// TIA Portal V20 export
FUNCTION_BLOCK "FB_IO_Device"   // FB4, LAD
{ S7_Optimized_Access := 'TRUE' }
// stored: MemoryReserve 100, SetENOAutomatically false
   VAR_INPUT
      Test_Station : SInt;
      Life_Trigger : Bool;
      Star_Test : Bool;
      Button_Start_Approve : Bool;
      Electrical_Current_Test_Approved : Bool;
      Visual_Test_Approved : Bool;
      Electrical_Current_Read : UInt;
      Electrical_Voltage_Read : UInt;
      In_Functional_Test : "IO_Device_Functinal_Test";
      In_Test_Parameters : "IO_Device_Test_Parameters";
   END_VAR
   VAR_OUTPUT
      Reset_Functional_Test : Bool;
      Out_Test_Parameters : "IO_Device_Test_Parameters";
      Out_Functional_Test : "IO_Device_Functinal_Test";
      Out_Electrical_Voltage_Read : UInt;
   END_VAR
   VAR_TEMP   // added for the SCL form of the ladder/FBD networks
      _w1 : Bool;
   END_VAR
BEGIN

REGION Network 1: Test Parameters
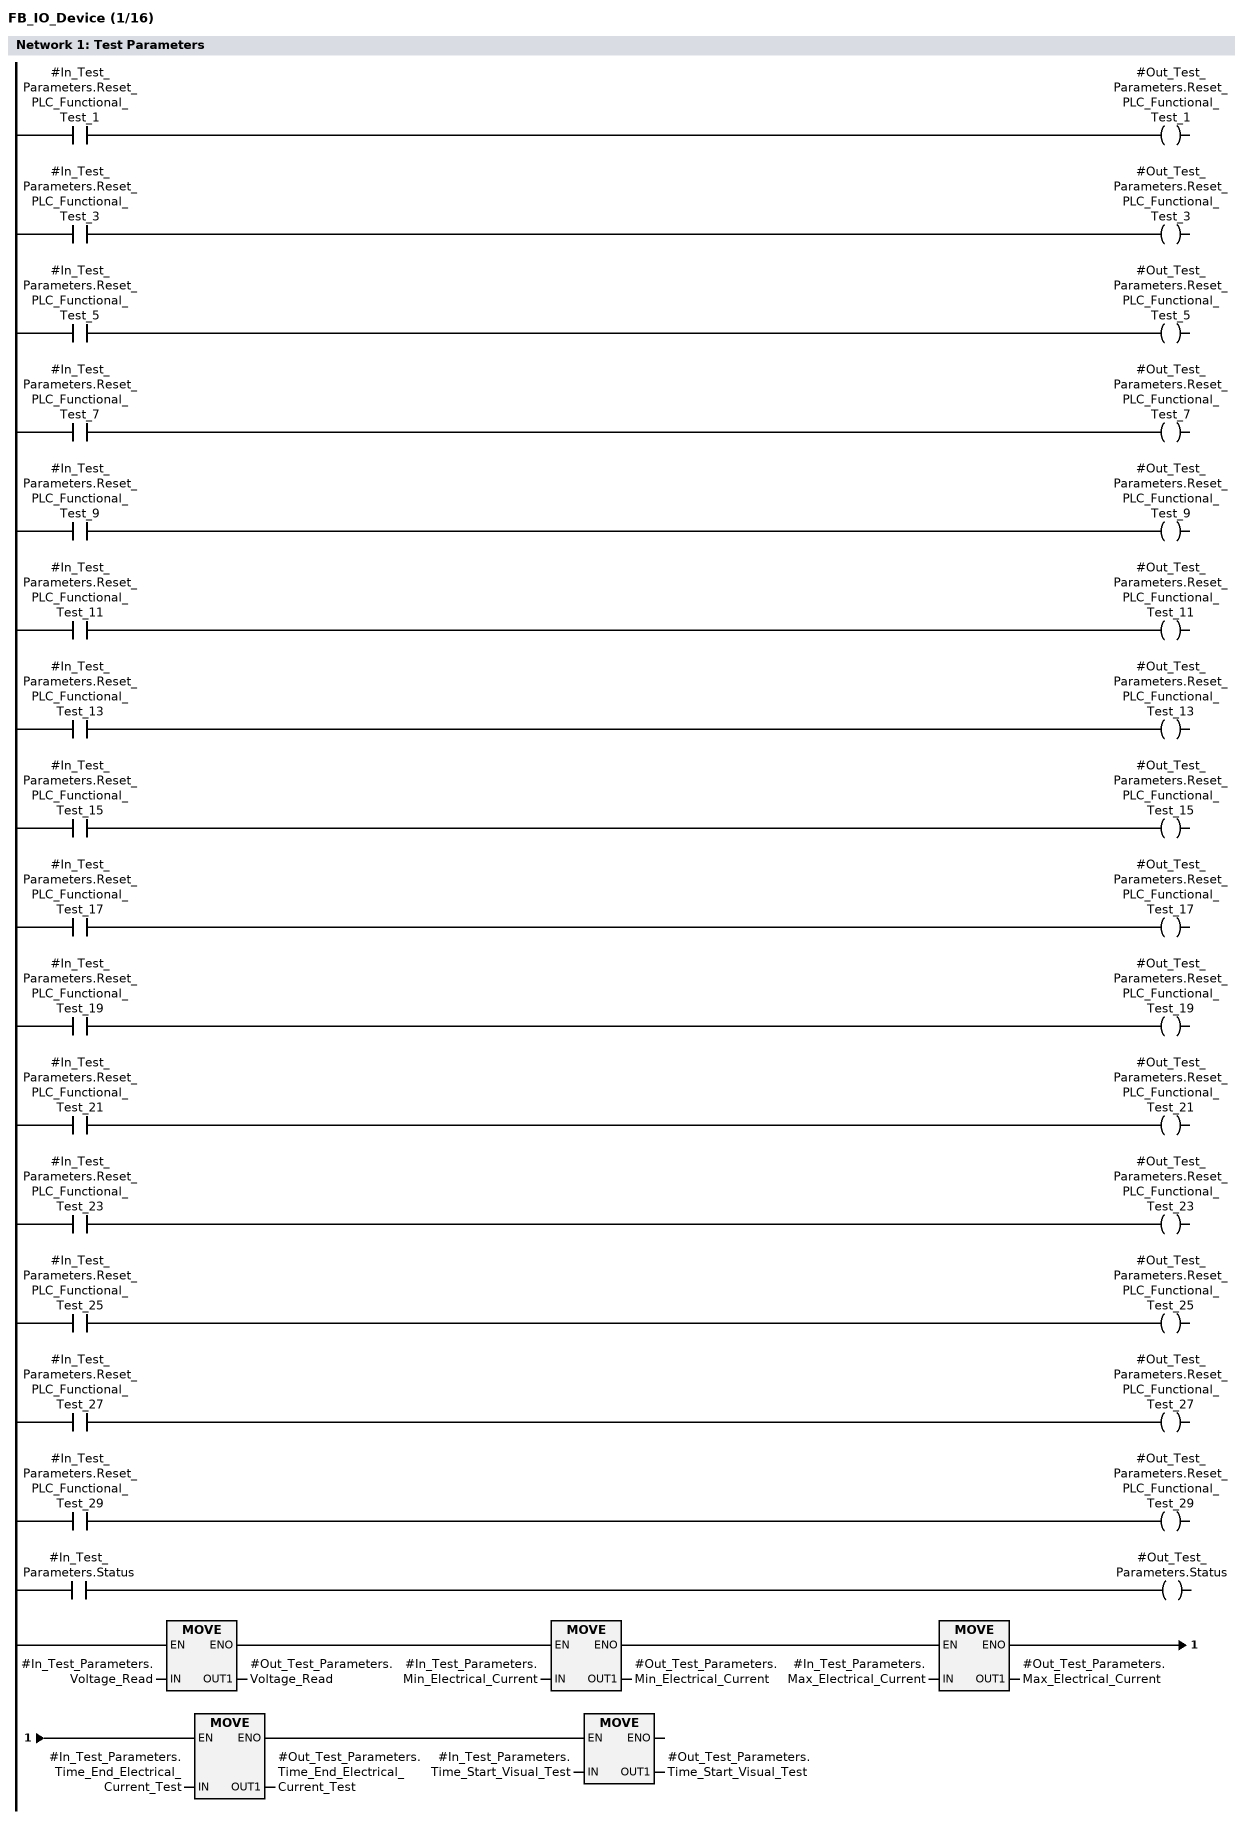
   RUNG wire#powerrail
      Contact( #In_Test_Parameters.Reset_PLC_Functional_Test_1 )
      Coil( #Out_Test_Parameters.Reset_PLC_Functional_Test_1 )
   END_RUNG
   RUNG wire#powerrail
      Contact( #In_Test_Parameters.Reset_PLC_Functional_Test_3 )
      Coil( #Out_Test_Parameters.Reset_PLC_Functional_Test_3 )
   END_RUNG
   RUNG wire#powerrail
      Contact( #In_Test_Parameters.Reset_PLC_Functional_Test_5 )
      Coil( #Out_Test_Parameters.Reset_PLC_Functional_Test_5 )
   END_RUNG
   RUNG wire#powerrail
      Contact( #In_Test_Parameters.Reset_PLC_Functional_Test_7 )
      Coil( #Out_Test_Parameters.Reset_PLC_Functional_Test_7 )
   END_RUNG
   RUNG wire#powerrail
      Contact( #In_Test_Parameters.Reset_PLC_Functional_Test_9 )
      Coil( #Out_Test_Parameters.Reset_PLC_Functional_Test_9 )
   END_RUNG
   RUNG wire#powerrail
      Contact( #In_Test_Parameters.Reset_PLC_Functional_Test_11 )
      Coil( #Out_Test_Parameters.Reset_PLC_Functional_Test_11 )
   END_RUNG
   RUNG wire#powerrail
      Contact( #In_Test_Parameters.Reset_PLC_Functional_Test_13 )
      Coil( #Out_Test_Parameters.Reset_PLC_Functional_Test_13 )
   END_RUNG
   RUNG wire#powerrail
      Contact( #In_Test_Parameters.Reset_PLC_Functional_Test_15 )
      Coil( #Out_Test_Parameters.Reset_PLC_Functional_Test_15 )
   END_RUNG
   RUNG wire#powerrail
      Contact( #In_Test_Parameters.Reset_PLC_Functional_Test_17 )
      Coil( #Out_Test_Parameters.Reset_PLC_Functional_Test_17 )
   END_RUNG
   RUNG wire#powerrail
      Contact( #In_Test_Parameters.Reset_PLC_Functional_Test_19 )
      Coil( #Out_Test_Parameters.Reset_PLC_Functional_Test_19 )
   END_RUNG
   RUNG wire#powerrail
      Contact( #In_Test_Parameters.Reset_PLC_Functional_Test_21 )
      Coil( #Out_Test_Parameters.Reset_PLC_Functional_Test_21 )
   END_RUNG
   RUNG wire#powerrail
      Contact( #In_Test_Parameters.Reset_PLC_Functional_Test_23 )
      Coil( #Out_Test_Parameters.Reset_PLC_Functional_Test_23 )
   END_RUNG
   RUNG wire#powerrail
      Contact( #In_Test_Parameters.Reset_PLC_Functional_Test_25 )
      Coil( #Out_Test_Parameters.Reset_PLC_Functional_Test_25 )
   END_RUNG
   RUNG wire#powerrail
      Contact( #In_Test_Parameters.Reset_PLC_Functional_Test_27 )
      Coil( #Out_Test_Parameters.Reset_PLC_Functional_Test_27 )
   END_RUNG
   RUNG wire#powerrail
      Contact( #In_Test_Parameters.Reset_PLC_Functional_Test_29 )
      Coil( #Out_Test_Parameters.Reset_PLC_Functional_Test_29 )
   END_RUNG
   RUNG wire#powerrail
      Contact( #In_Test_Parameters.Status )
      Coil( #Out_Test_Parameters.Status )
   END_RUNG
   RUNG wire#powerrail
      Move(in := #In_Test_Parameters.Voltage_Read, out1 => #Out_Test_Parameters.Voltage_Read)
      Move(in := #In_Test_Parameters.Min_Electrical_Current, out1 => #Out_Test_Parameters.Min_Electrical_Current)
      Move(in := #In_Test_Parameters.Max_Electrical_Current, out1 => #Out_Test_Parameters.Max_Electrical_Current)
      Move(in := #In_Test_Parameters.Time_End_Electrical_Current_Test, out1 => #Out_Test_Parameters.Time_End_Electrical_Current_Test)
      Move(in := #In_Test_Parameters.Time_Start_Visual_Test, out1 => #Out_Test_Parameters.Time_Start_Visual_Test)
   END_RUNG
   // the same network as SCL:
   #Out_Test_Parameters.Reset_PLC_Functional_Test_1 := #In_Test_Parameters.Reset_PLC_Functional_Test_1;
   #Out_Test_Parameters.Reset_PLC_Functional_Test_3 := #In_Test_Parameters.Reset_PLC_Functional_Test_3;
   #Out_Test_Parameters.Reset_PLC_Functional_Test_5 := #In_Test_Parameters.Reset_PLC_Functional_Test_5;
   #Out_Test_Parameters.Reset_PLC_Functional_Test_7 := #In_Test_Parameters.Reset_PLC_Functional_Test_7;
   #Out_Test_Parameters.Reset_PLC_Functional_Test_9 := #In_Test_Parameters.Reset_PLC_Functional_Test_9;
   #Out_Test_Parameters.Reset_PLC_Functional_Test_11 := #In_Test_Parameters.Reset_PLC_Functional_Test_11;
   #Out_Test_Parameters.Reset_PLC_Functional_Test_13 := #In_Test_Parameters.Reset_PLC_Functional_Test_13;
   #Out_Test_Parameters.Reset_PLC_Functional_Test_15 := #In_Test_Parameters.Reset_PLC_Functional_Test_15;
   #Out_Test_Parameters.Reset_PLC_Functional_Test_17 := #In_Test_Parameters.Reset_PLC_Functional_Test_17;
   #Out_Test_Parameters.Reset_PLC_Functional_Test_19 := #In_Test_Parameters.Reset_PLC_Functional_Test_19;
   #Out_Test_Parameters.Reset_PLC_Functional_Test_21 := #In_Test_Parameters.Reset_PLC_Functional_Test_21;
   #Out_Test_Parameters.Reset_PLC_Functional_Test_23 := #In_Test_Parameters.Reset_PLC_Functional_Test_23;
   #Out_Test_Parameters.Reset_PLC_Functional_Test_25 := #In_Test_Parameters.Reset_PLC_Functional_Test_25;
   #Out_Test_Parameters.Reset_PLC_Functional_Test_27 := #In_Test_Parameters.Reset_PLC_Functional_Test_27;
   #Out_Test_Parameters.Reset_PLC_Functional_Test_29 := #In_Test_Parameters.Reset_PLC_Functional_Test_29;
   #Out_Test_Parameters.Status := #In_Test_Parameters.Status;
   #Out_Test_Parameters.Voltage_Read := #In_Test_Parameters.Voltage_Read;
   #Out_Test_Parameters.Min_Electrical_Current := #In_Test_Parameters.Min_Electrical_Current;
   #Out_Test_Parameters.Max_Electrical_Current := #In_Test_Parameters.Max_Electrical_Current;
   #Out_Test_Parameters.Time_End_Electrical_Current_Test := #In_Test_Parameters.Time_End_Electrical_Current_Test;
   #Out_Test_Parameters.Time_Start_Visual_Test := #In_Test_Parameters.Time_Start_Visual_Test;
END_REGION

REGION Network 2: Functional Test Station 1
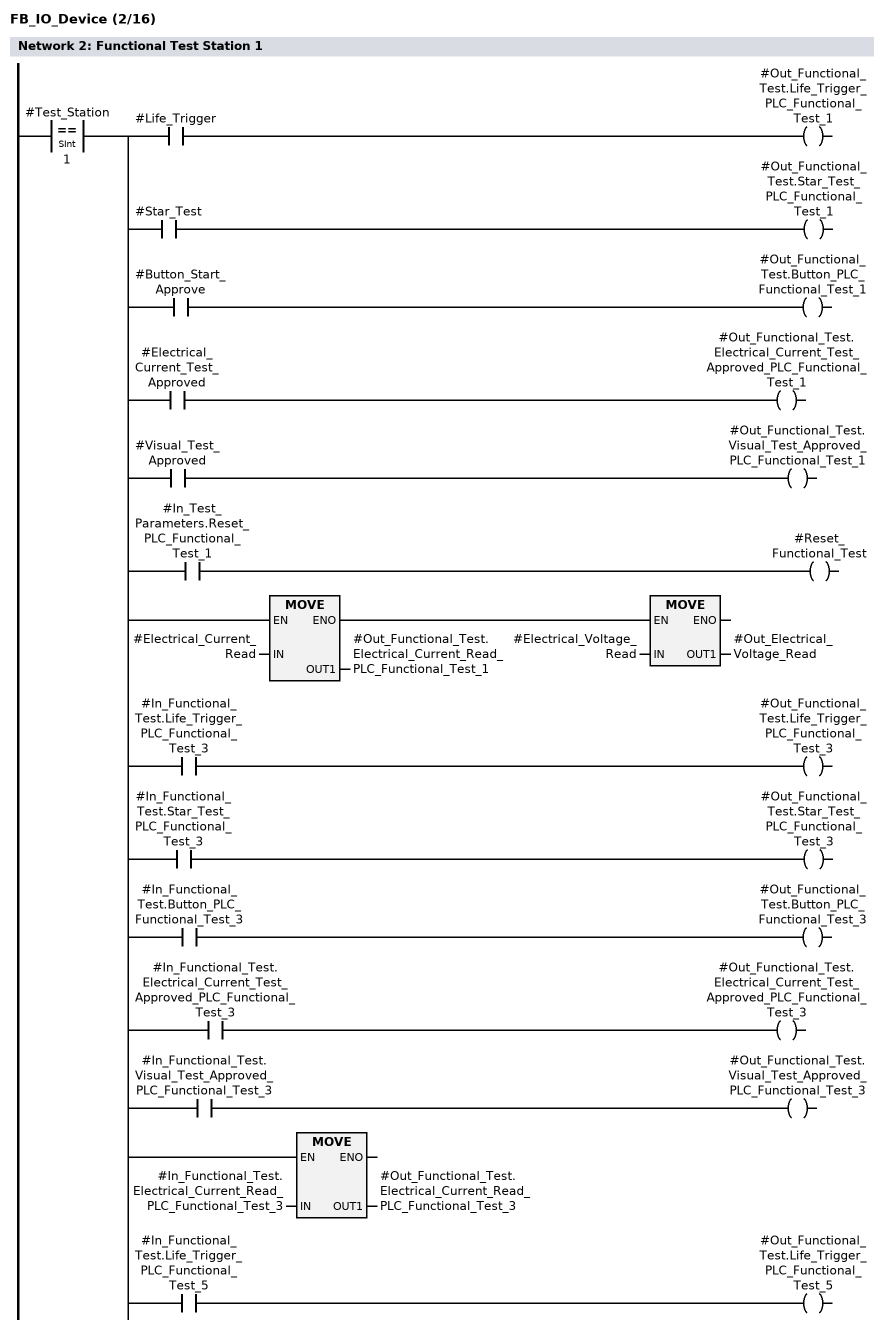
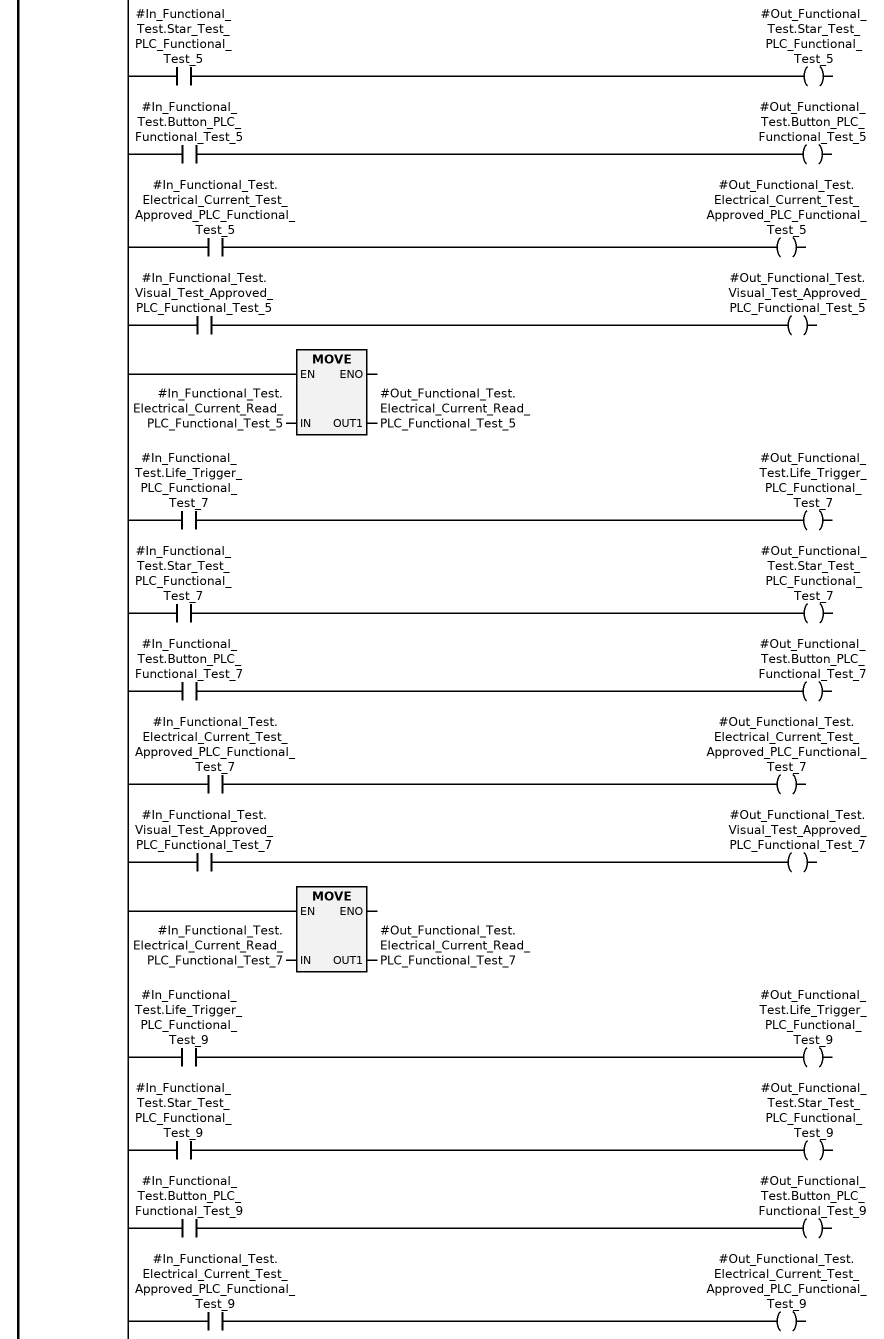
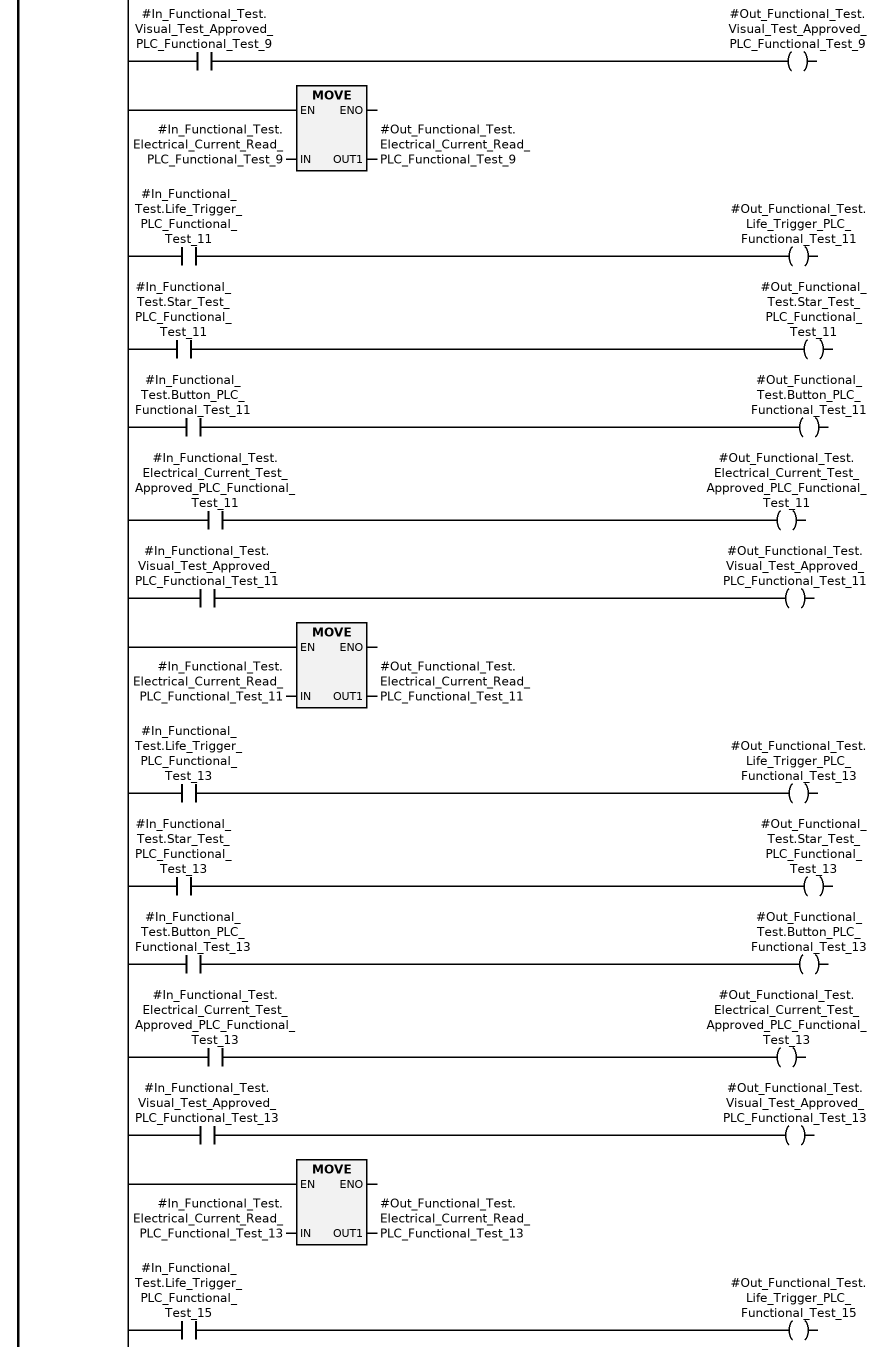
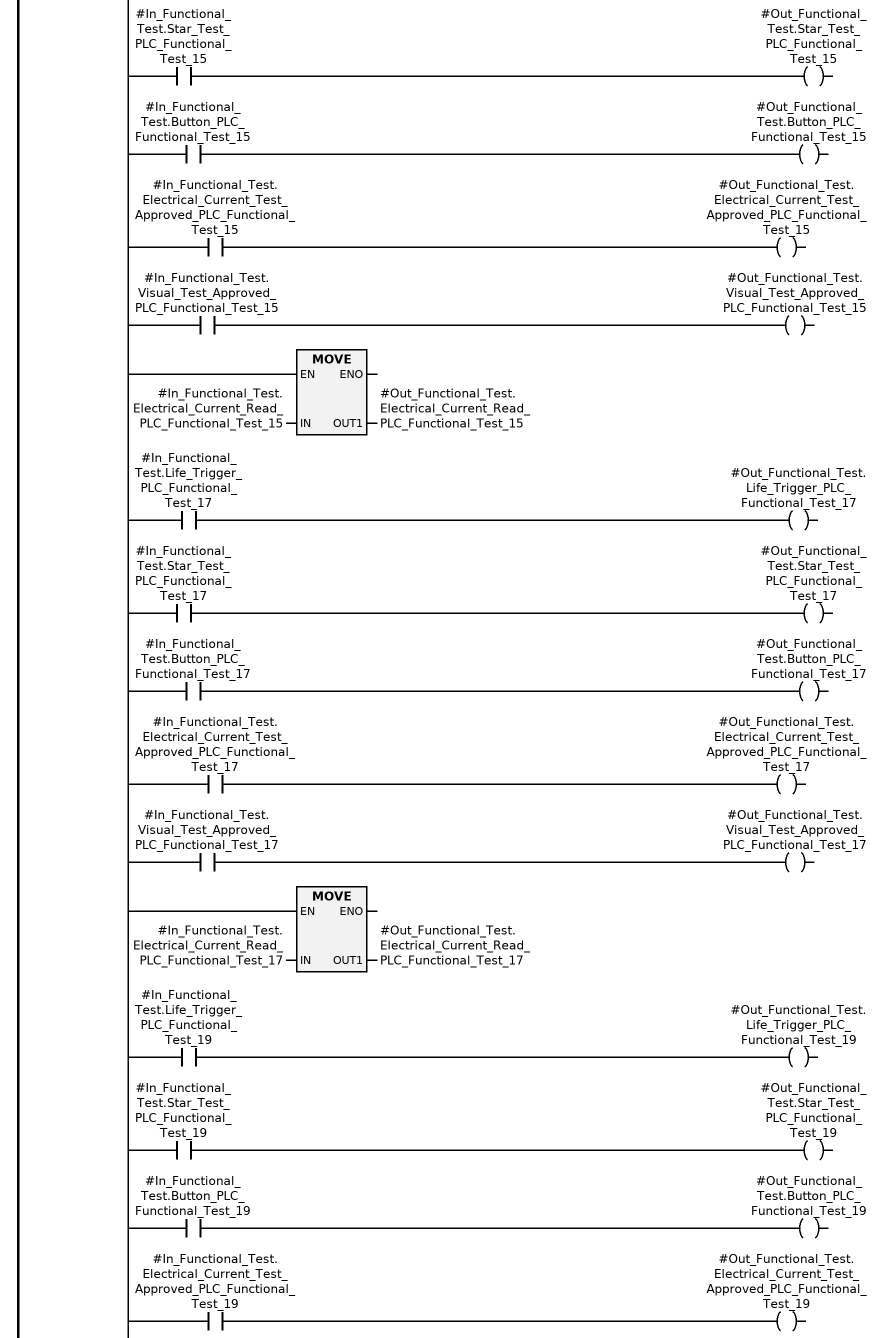
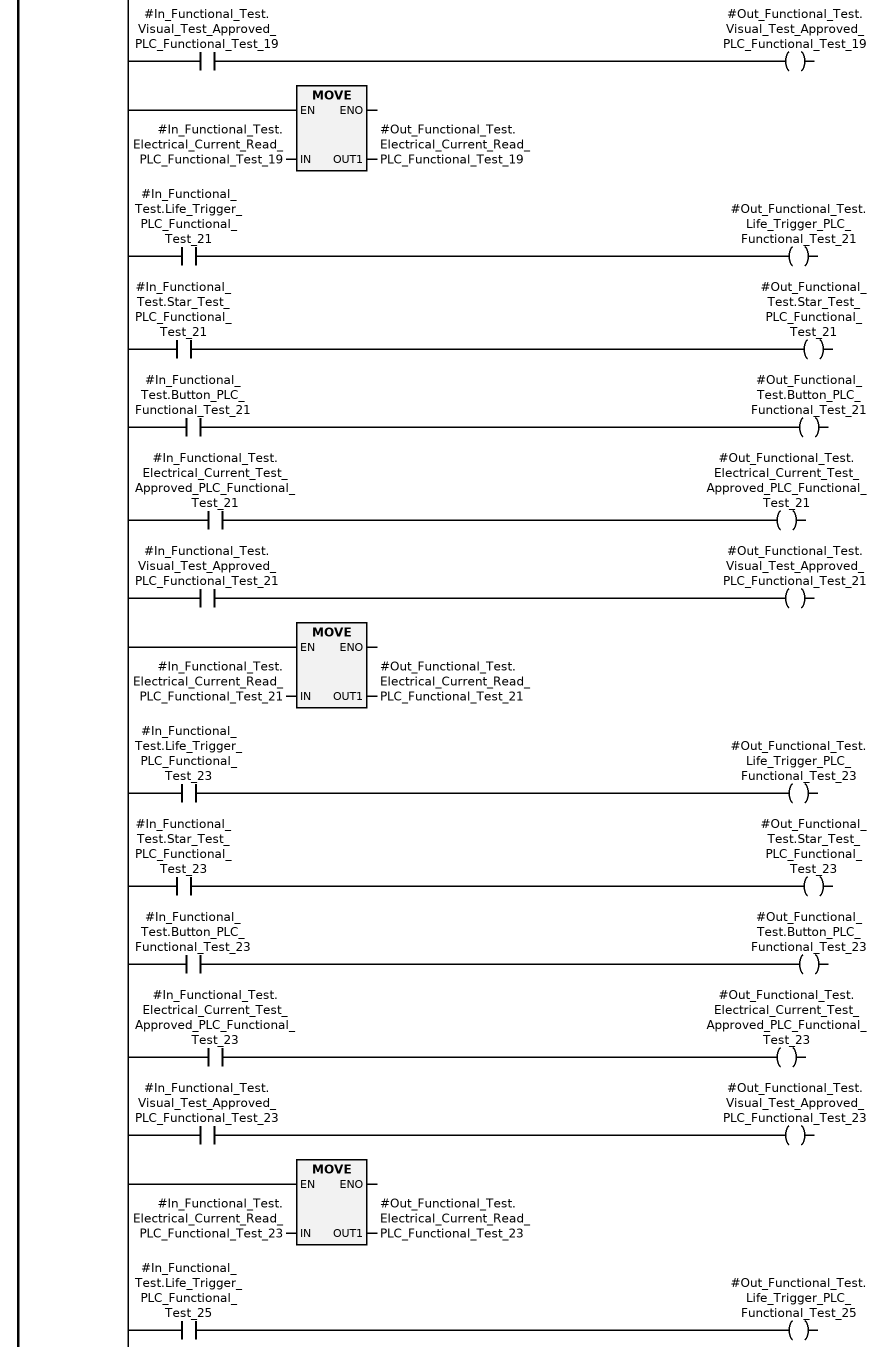
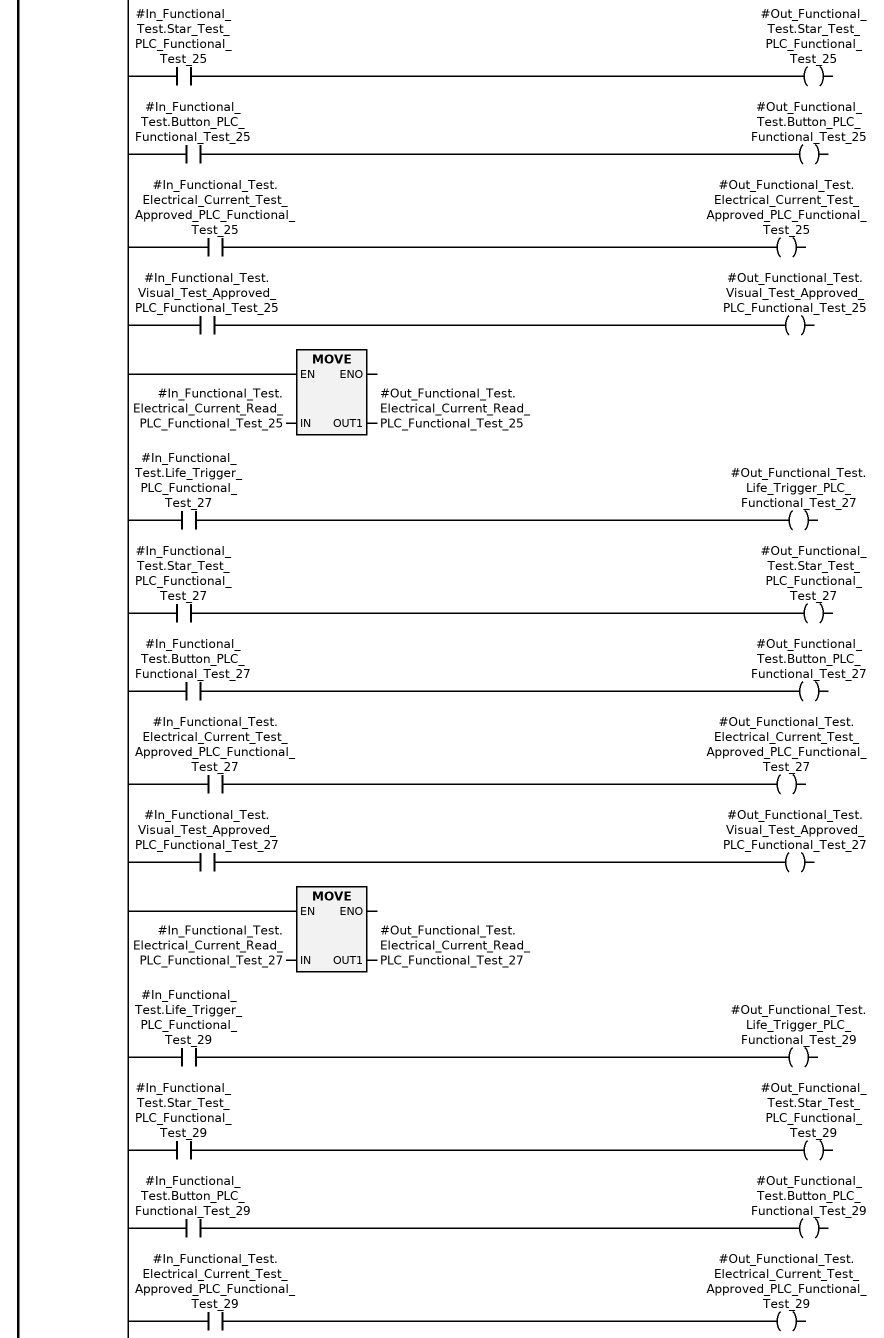
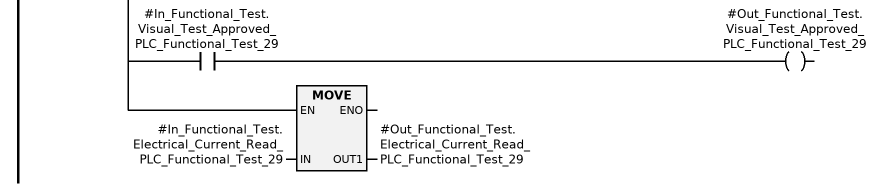
   RUNG wire#powerrail
      { S7_Templates := "SrcType := SInt" } EQ_Contact(in1 := #Test_Station, in2 := 1)
      wire#w1
      Contact( #Life_Trigger )
      Coil( #Out_Functional_Test.Life_Trigger_PLC_Functional_Test_1 )
   END_RUNG
   RUNG wire#w1
      Contact( #Star_Test )
      Coil( #Out_Functional_Test.Star_Test_PLC_Functional_Test_1 )
   END_RUNG
   RUNG wire#w1
      Contact( #Button_Start_Approve )
      Coil( #Out_Functional_Test.Button_PLC_Functional_Test_1 )
   END_RUNG
   RUNG wire#w1
      Contact( #Electrical_Current_Test_Approved )
      Coil( #Out_Functional_Test.Electrical_Current_Test_Approved_PLC_Functional_Test_1 )
   END_RUNG
   RUNG wire#w1
      Contact( #Visual_Test_Approved )
      Coil( #Out_Functional_Test.Visual_Test_Approved_PLC_Functional_Test_1 )
   END_RUNG
   RUNG wire#w1
      Contact( #In_Test_Parameters.Reset_PLC_Functional_Test_1 )
      Coil( #Reset_Functional_Test )
   END_RUNG
   RUNG wire#w1
      Move(in := #Electrical_Current_Read, out1 => #Out_Functional_Test.Electrical_Current_Read_PLC_Functional_Test_1)
      Move(in := #Electrical_Voltage_Read, out1 => #Out_Electrical_Voltage_Read)
   END_RUNG
   RUNG wire#w1
      Contact( #In_Functional_Test.Life_Trigger_PLC_Functional_Test_3 )
      Coil( #Out_Functional_Test.Life_Trigger_PLC_Functional_Test_3 )
   END_RUNG
   RUNG wire#w1
      Contact( #In_Functional_Test.Star_Test_PLC_Functional_Test_3 )
      Coil( #Out_Functional_Test.Star_Test_PLC_Functional_Test_3 )
   END_RUNG
   RUNG wire#w1
      Contact( #In_Functional_Test.Button_PLC_Functional_Test_3 )
      Coil( #Out_Functional_Test.Button_PLC_Functional_Test_3 )
   END_RUNG
   RUNG wire#w1
      Contact( #In_Functional_Test.Electrical_Current_Test_Approved_PLC_Functional_Test_3 )
      Coil( #Out_Functional_Test.Electrical_Current_Test_Approved_PLC_Functional_Test_3 )
   END_RUNG
   RUNG wire#w1
      Contact( #In_Functional_Test.Visual_Test_Approved_PLC_Functional_Test_3 )
      Coil( #Out_Functional_Test.Visual_Test_Approved_PLC_Functional_Test_3 )
   END_RUNG
   RUNG wire#w1
      Move(in := #In_Functional_Test.Electrical_Current_Read_PLC_Functional_Test_3, out1 => #Out_Functional_Test.Electrical_Current_Read_PLC_Functional_Test_3)
   END_RUNG
   RUNG wire#w1
      Contact( #In_Functional_Test.Life_Trigger_PLC_Functional_Test_5 )
      Coil( #Out_Functional_Test.Life_Trigger_PLC_Functional_Test_5 )
   END_RUNG
   RUNG wire#w1
      Contact( #In_Functional_Test.Star_Test_PLC_Functional_Test_5 )
      Coil( #Out_Functional_Test.Star_Test_PLC_Functional_Test_5 )
   END_RUNG
   RUNG wire#w1
      Contact( #In_Functional_Test.Button_PLC_Functional_Test_5 )
      Coil( #Out_Functional_Test.Button_PLC_Functional_Test_5 )
   END_RUNG
   RUNG wire#w1
      Contact( #In_Functional_Test.Electrical_Current_Test_Approved_PLC_Functional_Test_5 )
      Coil( #Out_Functional_Test.Electrical_Current_Test_Approved_PLC_Functional_Test_5 )
   END_RUNG
   RUNG wire#w1
      Contact( #In_Functional_Test.Visual_Test_Approved_PLC_Functional_Test_5 )
      Coil( #Out_Functional_Test.Visual_Test_Approved_PLC_Functional_Test_5 )
   END_RUNG
   RUNG wire#w1
      Move(in := #In_Functional_Test.Electrical_Current_Read_PLC_Functional_Test_5, out1 => #Out_Functional_Test.Electrical_Current_Read_PLC_Functional_Test_5)
   END_RUNG
   RUNG wire#w1
      Contact( #In_Functional_Test.Life_Trigger_PLC_Functional_Test_7 )
      Coil( #Out_Functional_Test.Life_Trigger_PLC_Functional_Test_7 )
   END_RUNG
   RUNG wire#w1
      Contact( #In_Functional_Test.Star_Test_PLC_Functional_Test_7 )
      Coil( #Out_Functional_Test.Star_Test_PLC_Functional_Test_7 )
   END_RUNG
   RUNG wire#w1
      Contact( #In_Functional_Test.Button_PLC_Functional_Test_7 )
      Coil( #Out_Functional_Test.Button_PLC_Functional_Test_7 )
   END_RUNG
   RUNG wire#w1
      Contact( #In_Functional_Test.Electrical_Current_Test_Approved_PLC_Functional_Test_7 )
      Coil( #Out_Functional_Test.Electrical_Current_Test_Approved_PLC_Functional_Test_7 )
   END_RUNG
   RUNG wire#w1
      Contact( #In_Functional_Test.Visual_Test_Approved_PLC_Functional_Test_7 )
      Coil( #Out_Functional_Test.Visual_Test_Approved_PLC_Functional_Test_7 )
   END_RUNG
   RUNG wire#w1
      Move(in := #In_Functional_Test.Electrical_Current_Read_PLC_Functional_Test_7, out1 => #Out_Functional_Test.Electrical_Current_Read_PLC_Functional_Test_7)
   END_RUNG
   RUNG wire#w1
      Contact( #In_Functional_Test.Life_Trigger_PLC_Functional_Test_9 )
      Coil( #Out_Functional_Test.Life_Trigger_PLC_Functional_Test_9 )
   END_RUNG
   RUNG wire#w1
      Contact( #In_Functional_Test.Star_Test_PLC_Functional_Test_9 )
      Coil( #Out_Functional_Test.Star_Test_PLC_Functional_Test_9 )
   END_RUNG
   RUNG wire#w1
      Contact( #In_Functional_Test.Button_PLC_Functional_Test_9 )
      Coil( #Out_Functional_Test.Button_PLC_Functional_Test_9 )
   END_RUNG
   RUNG wire#w1
      Contact( #In_Functional_Test.Electrical_Current_Test_Approved_PLC_Functional_Test_9 )
      Coil( #Out_Functional_Test.Electrical_Current_Test_Approved_PLC_Functional_Test_9 )
   END_RUNG
   RUNG wire#w1
      Contact( #In_Functional_Test.Visual_Test_Approved_PLC_Functional_Test_9 )
      Coil( #Out_Functional_Test.Visual_Test_Approved_PLC_Functional_Test_9 )
   END_RUNG
   RUNG wire#w1
      Move(in := #In_Functional_Test.Electrical_Current_Read_PLC_Functional_Test_9, out1 => #Out_Functional_Test.Electrical_Current_Read_PLC_Functional_Test_9)
   END_RUNG
   RUNG wire#w1
      Contact( #In_Functional_Test.Life_Trigger_PLC_Functional_Test_11 )
      Coil( #Out_Functional_Test.Life_Trigger_PLC_Functional_Test_11 )
   END_RUNG
   RUNG wire#w1
      Contact( #In_Functional_Test.Star_Test_PLC_Functional_Test_11 )
      Coil( #Out_Functional_Test.Star_Test_PLC_Functional_Test_11 )
   END_RUNG
   RUNG wire#w1
      Contact( #In_Functional_Test.Button_PLC_Functional_Test_11 )
      Coil( #Out_Functional_Test.Button_PLC_Functional_Test_11 )
   END_RUNG
   RUNG wire#w1
      Contact( #In_Functional_Test.Electrical_Current_Test_Approved_PLC_Functional_Test_11 )
      Coil( #Out_Functional_Test.Electrical_Current_Test_Approved_PLC_Functional_Test_11 )
   END_RUNG
   RUNG wire#w1
      Contact( #In_Functional_Test.Visual_Test_Approved_PLC_Functional_Test_11 )
      Coil( #Out_Functional_Test.Visual_Test_Approved_PLC_Functional_Test_11 )
   END_RUNG
   RUNG wire#w1
      Move(in := #In_Functional_Test.Electrical_Current_Read_PLC_Functional_Test_11, out1 => #Out_Functional_Test.Electrical_Current_Read_PLC_Functional_Test_11)
   END_RUNG
   RUNG wire#w1
      Contact( #In_Functional_Test.Life_Trigger_PLC_Functional_Test_13 )
      Coil( #Out_Functional_Test.Life_Trigger_PLC_Functional_Test_13 )
   END_RUNG
   RUNG wire#w1
      Contact( #In_Functional_Test.Star_Test_PLC_Functional_Test_13 )
      Coil( #Out_Functional_Test.Star_Test_PLC_Functional_Test_13 )
   END_RUNG
   RUNG wire#w1
      Contact( #In_Functional_Test.Button_PLC_Functional_Test_13 )
      Coil( #Out_Functional_Test.Button_PLC_Functional_Test_13 )
   END_RUNG
   RUNG wire#w1
      Contact( #In_Functional_Test.Electrical_Current_Test_Approved_PLC_Functional_Test_13 )
      Coil( #Out_Functional_Test.Electrical_Current_Test_Approved_PLC_Functional_Test_13 )
   END_RUNG
   RUNG wire#w1
      Contact( #In_Functional_Test.Visual_Test_Approved_PLC_Functional_Test_13 )
      Coil( #Out_Functional_Test.Visual_Test_Approved_PLC_Functional_Test_13 )
   END_RUNG
   RUNG wire#w1
      Move(in := #In_Functional_Test.Electrical_Current_Read_PLC_Functional_Test_13, out1 => #Out_Functional_Test.Electrical_Current_Read_PLC_Functional_Test_13)
   END_RUNG
   RUNG wire#w1
      Contact( #In_Functional_Test.Life_Trigger_PLC_Functional_Test_15 )
      Coil( #Out_Functional_Test.Life_Trigger_PLC_Functional_Test_15 )
   END_RUNG
   RUNG wire#w1
      Contact( #In_Functional_Test.Star_Test_PLC_Functional_Test_15 )
      Coil( #Out_Functional_Test.Star_Test_PLC_Functional_Test_15 )
   END_RUNG
   RUNG wire#w1
      Contact( #In_Functional_Test.Button_PLC_Functional_Test_15 )
      Coil( #Out_Functional_Test.Button_PLC_Functional_Test_15 )
   END_RUNG
   RUNG wire#w1
      Contact( #In_Functional_Test.Electrical_Current_Test_Approved_PLC_Functional_Test_15 )
      Coil( #Out_Functional_Test.Electrical_Current_Test_Approved_PLC_Functional_Test_15 )
   END_RUNG
   RUNG wire#w1
      Contact( #In_Functional_Test.Visual_Test_Approved_PLC_Functional_Test_15 )
      Coil( #Out_Functional_Test.Visual_Test_Approved_PLC_Functional_Test_15 )
   END_RUNG
   RUNG wire#w1
      Move(in := #In_Functional_Test.Electrical_Current_Read_PLC_Functional_Test_15, out1 => #Out_Functional_Test.Electrical_Current_Read_PLC_Functional_Test_15)
   END_RUNG
   RUNG wire#w1
      Contact( #In_Functional_Test.Life_Trigger_PLC_Functional_Test_17 )
      Coil( #Out_Functional_Test.Life_Trigger_PLC_Functional_Test_17 )
   END_RUNG
   RUNG wire#w1
      Contact( #In_Functional_Test.Star_Test_PLC_Functional_Test_17 )
      Coil( #Out_Functional_Test.Star_Test_PLC_Functional_Test_17 )
   END_RUNG
   RUNG wire#w1
      Contact( #In_Functional_Test.Button_PLC_Functional_Test_17 )
      Coil( #Out_Functional_Test.Button_PLC_Functional_Test_17 )
   END_RUNG
   RUNG wire#w1
      Contact( #In_Functional_Test.Electrical_Current_Test_Approved_PLC_Functional_Test_17 )
      Coil( #Out_Functional_Test.Electrical_Current_Test_Approved_PLC_Functional_Test_17 )
   END_RUNG
   RUNG wire#w1
      Contact( #In_Functional_Test.Visual_Test_Approved_PLC_Functional_Test_17 )
      Coil( #Out_Functional_Test.Visual_Test_Approved_PLC_Functional_Test_17 )
   END_RUNG
   RUNG wire#w1
      Move(in := #In_Functional_Test.Electrical_Current_Read_PLC_Functional_Test_17, out1 => #Out_Functional_Test.Electrical_Current_Read_PLC_Functional_Test_17)
   END_RUNG
   RUNG wire#w1
      Contact( #In_Functional_Test.Life_Trigger_PLC_Functional_Test_19 )
      Coil( #Out_Functional_Test.Life_Trigger_PLC_Functional_Test_19 )
   END_RUNG
   RUNG wire#w1
      Contact( #In_Functional_Test.Star_Test_PLC_Functional_Test_19 )
      Coil( #Out_Functional_Test.Star_Test_PLC_Functional_Test_19 )
   END_RUNG
   RUNG wire#w1
      Contact( #In_Functional_Test.Button_PLC_Functional_Test_19 )
      Coil( #Out_Functional_Test.Button_PLC_Functional_Test_19 )
   END_RUNG
   RUNG wire#w1
      Contact( #In_Functional_Test.Electrical_Current_Test_Approved_PLC_Functional_Test_19 )
      Coil( #Out_Functional_Test.Electrical_Current_Test_Approved_PLC_Functional_Test_19 )
   END_RUNG
   RUNG wire#w1
      Contact( #In_Functional_Test.Visual_Test_Approved_PLC_Functional_Test_19 )
      Coil( #Out_Functional_Test.Visual_Test_Approved_PLC_Functional_Test_19 )
   END_RUNG
   RUNG wire#w1
      Move(in := #In_Functional_Test.Electrical_Current_Read_PLC_Functional_Test_19, out1 => #Out_Functional_Test.Electrical_Current_Read_PLC_Functional_Test_19)
   END_RUNG
   RUNG wire#w1
      Contact( #In_Functional_Test.Life_Trigger_PLC_Functional_Test_21 )
      Coil( #Out_Functional_Test.Life_Trigger_PLC_Functional_Test_21 )
   END_RUNG
   RUNG wire#w1
      Contact( #In_Functional_Test.Star_Test_PLC_Functional_Test_21 )
      Coil( #Out_Functional_Test.Star_Test_PLC_Functional_Test_21 )
   END_RUNG
   RUNG wire#w1
      Contact( #In_Functional_Test.Button_PLC_Functional_Test_21 )
      Coil( #Out_Functional_Test.Button_PLC_Functional_Test_21 )
   END_RUNG
   RUNG wire#w1
      Contact( #In_Functional_Test.Electrical_Current_Test_Approved_PLC_Functional_Test_21 )
      Coil( #Out_Functional_Test.Electrical_Current_Test_Approved_PLC_Functional_Test_21 )
   END_RUNG
   RUNG wire#w1
      Contact( #In_Functional_Test.Visual_Test_Approved_PLC_Functional_Test_21 )
      Coil( #Out_Functional_Test.Visual_Test_Approved_PLC_Functional_Test_21 )
   END_RUNG
   RUNG wire#w1
      Move(in := #In_Functional_Test.Electrical_Current_Read_PLC_Functional_Test_21, out1 => #Out_Functional_Test.Electrical_Current_Read_PLC_Functional_Test_21)
   END_RUNG
   RUNG wire#w1
      Contact( #In_Functional_Test.Life_Trigger_PLC_Functional_Test_23 )
      Coil( #Out_Functional_Test.Life_Trigger_PLC_Functional_Test_23 )
   END_RUNG
   RUNG wire#w1
      Contact( #In_Functional_Test.Star_Test_PLC_Functional_Test_23 )
      Coil( #Out_Functional_Test.Star_Test_PLC_Functional_Test_23 )
   END_RUNG
   RUNG wire#w1
      Contact( #In_Functional_Test.Button_PLC_Functional_Test_23 )
      Coil( #Out_Functional_Test.Button_PLC_Functional_Test_23 )
   END_RUNG
   RUNG wire#w1
      Contact( #In_Functional_Test.Electrical_Current_Test_Approved_PLC_Functional_Test_23 )
      Coil( #Out_Functional_Test.Electrical_Current_Test_Approved_PLC_Functional_Test_23 )
   END_RUNG
   RUNG wire#w1
      Contact( #In_Functional_Test.Visual_Test_Approved_PLC_Functional_Test_23 )
      Coil( #Out_Functional_Test.Visual_Test_Approved_PLC_Functional_Test_23 )
   END_RUNG
   RUNG wire#w1
      Move(in := #In_Functional_Test.Electrical_Current_Read_PLC_Functional_Test_23, out1 => #Out_Functional_Test.Electrical_Current_Read_PLC_Functional_Test_23)
   END_RUNG
   RUNG wire#w1
      Contact( #In_Functional_Test.Life_Trigger_PLC_Functional_Test_25 )
      Coil( #Out_Functional_Test.Life_Trigger_PLC_Functional_Test_25 )
   END_RUNG
   RUNG wire#w1
      Contact( #In_Functional_Test.Star_Test_PLC_Functional_Test_25 )
      Coil( #Out_Functional_Test.Star_Test_PLC_Functional_Test_25 )
   END_RUNG
   RUNG wire#w1
      Contact( #In_Functional_Test.Button_PLC_Functional_Test_25 )
      Coil( #Out_Functional_Test.Button_PLC_Functional_Test_25 )
   END_RUNG
   RUNG wire#w1
      Contact( #In_Functional_Test.Electrical_Current_Test_Approved_PLC_Functional_Test_25 )
      Coil( #Out_Functional_Test.Electrical_Current_Test_Approved_PLC_Functional_Test_25 )
   END_RUNG
   RUNG wire#w1
      Contact( #In_Functional_Test.Visual_Test_Approved_PLC_Functional_Test_25 )
      Coil( #Out_Functional_Test.Visual_Test_Approved_PLC_Functional_Test_25 )
   END_RUNG
   RUNG wire#w1
      Move(in := #In_Functional_Test.Electrical_Current_Read_PLC_Functional_Test_25, out1 => #Out_Functional_Test.Electrical_Current_Read_PLC_Functional_Test_25)
   END_RUNG
   RUNG wire#w1
      Contact( #In_Functional_Test.Life_Trigger_PLC_Functional_Test_27 )
      Coil( #Out_Functional_Test.Life_Trigger_PLC_Functional_Test_27 )
   END_RUNG
   RUNG wire#w1
      Contact( #In_Functional_Test.Star_Test_PLC_Functional_Test_27 )
      Coil( #Out_Functional_Test.Star_Test_PLC_Functional_Test_27 )
   END_RUNG
   RUNG wire#w1
      Contact( #In_Functional_Test.Button_PLC_Functional_Test_27 )
      Coil( #Out_Functional_Test.Button_PLC_Functional_Test_27 )
   END_RUNG
   RUNG wire#w1
      Contact( #In_Functional_Test.Electrical_Current_Test_Approved_PLC_Functional_Test_27 )
      Coil( #Out_Functional_Test.Electrical_Current_Test_Approved_PLC_Functional_Test_27 )
   END_RUNG
   RUNG wire#w1
      Contact( #In_Functional_Test.Visual_Test_Approved_PLC_Functional_Test_27 )
      Coil( #Out_Functional_Test.Visual_Test_Approved_PLC_Functional_Test_27 )
   END_RUNG
   RUNG wire#w1
      Move(in := #In_Functional_Test.Electrical_Current_Read_PLC_Functional_Test_27, out1 => #Out_Functional_Test.Electrical_Current_Read_PLC_Functional_Test_27)
   END_RUNG
   RUNG wire#w1
      Contact( #In_Functional_Test.Life_Trigger_PLC_Functional_Test_29 )
      Coil( #Out_Functional_Test.Life_Trigger_PLC_Functional_Test_29 )
   END_RUNG
   RUNG wire#w1
      Contact( #In_Functional_Test.Star_Test_PLC_Functional_Test_29 )
      Coil( #Out_Functional_Test.Star_Test_PLC_Functional_Test_29 )
   END_RUNG
   RUNG wire#w1
      Contact( #In_Functional_Test.Button_PLC_Functional_Test_29 )
      Coil( #Out_Functional_Test.Button_PLC_Functional_Test_29 )
   END_RUNG
   RUNG wire#w1
      Contact( #In_Functional_Test.Electrical_Current_Test_Approved_PLC_Functional_Test_29 )
      Coil( #Out_Functional_Test.Electrical_Current_Test_Approved_PLC_Functional_Test_29 )
   END_RUNG
   RUNG wire#w1
      Contact( #In_Functional_Test.Visual_Test_Approved_PLC_Functional_Test_29 )
      Coil( #Out_Functional_Test.Visual_Test_Approved_PLC_Functional_Test_29 )
   END_RUNG
   RUNG wire#w1
      Move(in := #In_Functional_Test.Electrical_Current_Read_PLC_Functional_Test_29, out1 => #Out_Functional_Test.Electrical_Current_Read_PLC_Functional_Test_29)
   END_RUNG
   // the same network as SCL:
   #_w1 := #Test_Station = 1;
   #Out_Functional_Test.Life_Trigger_PLC_Functional_Test_1 := #_w1 AND #Life_Trigger;
   #Out_Functional_Test.Star_Test_PLC_Functional_Test_1 := #_w1 AND #Star_Test;
   #Out_Functional_Test.Button_PLC_Functional_Test_1 := #_w1 AND #Button_Start_Approve;
   #Out_Functional_Test.Electrical_Current_Test_Approved_PLC_Functional_Test_1 := #_w1 AND #Electrical_Current_Test_Approved;
   #Out_Functional_Test.Visual_Test_Approved_PLC_Functional_Test_1 := #_w1 AND #Visual_Test_Approved;
   #Reset_Functional_Test := #_w1 AND #In_Test_Parameters.Reset_PLC_Functional_Test_1;
   IF #_w1 THEN
       #Out_Functional_Test.Electrical_Current_Read_PLC_Functional_Test_1 := #Electrical_Current_Read;
       #Out_Electrical_Voltage_Read := #Electrical_Voltage_Read;
   END_IF;
   #Out_Functional_Test.Life_Trigger_PLC_Functional_Test_3 := #_w1 AND #In_Functional_Test.Life_Trigger_PLC_Functional_Test_3;
   #Out_Functional_Test.Star_Test_PLC_Functional_Test_3 := #_w1 AND #In_Functional_Test.Star_Test_PLC_Functional_Test_3;
   #Out_Functional_Test.Button_PLC_Functional_Test_3 := #_w1 AND #In_Functional_Test.Button_PLC_Functional_Test_3;
   #Out_Functional_Test.Electrical_Current_Test_Approved_PLC_Functional_Test_3 := #_w1 AND #In_Functional_Test.Electrical_Current_Test_Approved_PLC_Functional_Test_3;
   #Out_Functional_Test.Visual_Test_Approved_PLC_Functional_Test_3 := #_w1 AND #In_Functional_Test.Visual_Test_Approved_PLC_Functional_Test_3;
   IF #_w1 THEN
       #Out_Functional_Test.Electrical_Current_Read_PLC_Functional_Test_3 := #In_Functional_Test.Electrical_Current_Read_PLC_Functional_Test_3;
   END_IF;
   #Out_Functional_Test.Life_Trigger_PLC_Functional_Test_5 := #_w1 AND #In_Functional_Test.Life_Trigger_PLC_Functional_Test_5;
   #Out_Functional_Test.Star_Test_PLC_Functional_Test_5 := #_w1 AND #In_Functional_Test.Star_Test_PLC_Functional_Test_5;
   #Out_Functional_Test.Button_PLC_Functional_Test_5 := #_w1 AND #In_Functional_Test.Button_PLC_Functional_Test_5;
   #Out_Functional_Test.Electrical_Current_Test_Approved_PLC_Functional_Test_5 := #_w1 AND #In_Functional_Test.Electrical_Current_Test_Approved_PLC_Functional_Test_5;
   #Out_Functional_Test.Visual_Test_Approved_PLC_Functional_Test_5 := #_w1 AND #In_Functional_Test.Visual_Test_Approved_PLC_Functional_Test_5;
   IF #_w1 THEN
       #Out_Functional_Test.Electrical_Current_Read_PLC_Functional_Test_5 := #In_Functional_Test.Electrical_Current_Read_PLC_Functional_Test_5;
   END_IF;
   #Out_Functional_Test.Life_Trigger_PLC_Functional_Test_7 := #_w1 AND #In_Functional_Test.Life_Trigger_PLC_Functional_Test_7;
   #Out_Functional_Test.Star_Test_PLC_Functional_Test_7 := #_w1 AND #In_Functional_Test.Star_Test_PLC_Functional_Test_7;
   #Out_Functional_Test.Button_PLC_Functional_Test_7 := #_w1 AND #In_Functional_Test.Button_PLC_Functional_Test_7;
   #Out_Functional_Test.Electrical_Current_Test_Approved_PLC_Functional_Test_7 := #_w1 AND #In_Functional_Test.Electrical_Current_Test_Approved_PLC_Functional_Test_7;
   #Out_Functional_Test.Visual_Test_Approved_PLC_Functional_Test_7 := #_w1 AND #In_Functional_Test.Visual_Test_Approved_PLC_Functional_Test_7;
   IF #_w1 THEN
       #Out_Functional_Test.Electrical_Current_Read_PLC_Functional_Test_7 := #In_Functional_Test.Electrical_Current_Read_PLC_Functional_Test_7;
   END_IF;
   #Out_Functional_Test.Life_Trigger_PLC_Functional_Test_9 := #_w1 AND #In_Functional_Test.Life_Trigger_PLC_Functional_Test_9;
   #Out_Functional_Test.Star_Test_PLC_Functional_Test_9 := #_w1 AND #In_Functional_Test.Star_Test_PLC_Functional_Test_9;
   #Out_Functional_Test.Button_PLC_Functional_Test_9 := #_w1 AND #In_Functional_Test.Button_PLC_Functional_Test_9;
   #Out_Functional_Test.Electrical_Current_Test_Approved_PLC_Functional_Test_9 := #_w1 AND #In_Functional_Test.Electrical_Current_Test_Approved_PLC_Functional_Test_9;
   #Out_Functional_Test.Visual_Test_Approved_PLC_Functional_Test_9 := #_w1 AND #In_Functional_Test.Visual_Test_Approved_PLC_Functional_Test_9;
   IF #_w1 THEN
       #Out_Functional_Test.Electrical_Current_Read_PLC_Functional_Test_9 := #In_Functional_Test.Electrical_Current_Read_PLC_Functional_Test_9;
   END_IF;
   #Out_Functional_Test.Life_Trigger_PLC_Functional_Test_11 := #_w1 AND #In_Functional_Test.Life_Trigger_PLC_Functional_Test_11;
   #Out_Functional_Test.Star_Test_PLC_Functional_Test_11 := #_w1 AND #In_Functional_Test.Star_Test_PLC_Functional_Test_11;
   #Out_Functional_Test.Button_PLC_Functional_Test_11 := #_w1 AND #In_Functional_Test.Button_PLC_Functional_Test_11;
   #Out_Functional_Test.Electrical_Current_Test_Approved_PLC_Functional_Test_11 := #_w1 AND #In_Functional_Test.Electrical_Current_Test_Approved_PLC_Functional_Test_11;
   #Out_Functional_Test.Visual_Test_Approved_PLC_Functional_Test_11 := #_w1 AND #In_Functional_Test.Visual_Test_Approved_PLC_Functional_Test_11;
   IF #_w1 THEN
       #Out_Functional_Test.Electrical_Current_Read_PLC_Functional_Test_11 := #In_Functional_Test.Electrical_Current_Read_PLC_Functional_Test_11;
   END_IF;
   #Out_Functional_Test.Life_Trigger_PLC_Functional_Test_13 := #_w1 AND #In_Functional_Test.Life_Trigger_PLC_Functional_Test_13;
   #Out_Functional_Test.Star_Test_PLC_Functional_Test_13 := #_w1 AND #In_Functional_Test.Star_Test_PLC_Functional_Test_13;
   #Out_Functional_Test.Button_PLC_Functional_Test_13 := #_w1 AND #In_Functional_Test.Button_PLC_Functional_Test_13;
   #Out_Functional_Test.Electrical_Current_Test_Approved_PLC_Functional_Test_13 := #_w1 AND #In_Functional_Test.Electrical_Current_Test_Approved_PLC_Functional_Test_13;
   #Out_Functional_Test.Visual_Test_Approved_PLC_Functional_Test_13 := #_w1 AND #In_Functional_Test.Visual_Test_Approved_PLC_Functional_Test_13;
   IF #_w1 THEN
       #Out_Functional_Test.Electrical_Current_Read_PLC_Functional_Test_13 := #In_Functional_Test.Electrical_Current_Read_PLC_Functional_Test_13;
   END_IF;
   #Out_Functional_Test.Life_Trigger_PLC_Functional_Test_15 := #_w1 AND #In_Functional_Test.Life_Trigger_PLC_Functional_Test_15;
   #Out_Functional_Test.Star_Test_PLC_Functional_Test_15 := #_w1 AND #In_Functional_Test.Star_Test_PLC_Functional_Test_15;
   #Out_Functional_Test.Button_PLC_Functional_Test_15 := #_w1 AND #In_Functional_Test.Button_PLC_Functional_Test_15;
   #Out_Functional_Test.Electrical_Current_Test_Approved_PLC_Functional_Test_15 := #_w1 AND #In_Functional_Test.Electrical_Current_Test_Approved_PLC_Functional_Test_15;
   #Out_Functional_Test.Visual_Test_Approved_PLC_Functional_Test_15 := #_w1 AND #In_Functional_Test.Visual_Test_Approved_PLC_Functional_Test_15;
   IF #_w1 THEN
       #Out_Functional_Test.Electrical_Current_Read_PLC_Functional_Test_15 := #In_Functional_Test.Electrical_Current_Read_PLC_Functional_Test_15;
   END_IF;
   #Out_Functional_Test.Life_Trigger_PLC_Functional_Test_17 := #_w1 AND #In_Functional_Test.Life_Trigger_PLC_Functional_Test_17;
   #Out_Functional_Test.Star_Test_PLC_Functional_Test_17 := #_w1 AND #In_Functional_Test.Star_Test_PLC_Functional_Test_17;
   #Out_Functional_Test.Button_PLC_Functional_Test_17 := #_w1 AND #In_Functional_Test.Button_PLC_Functional_Test_17;
   #Out_Functional_Test.Electrical_Current_Test_Approved_PLC_Functional_Test_17 := #_w1 AND #In_Functional_Test.Electrical_Current_Test_Approved_PLC_Functional_Test_17;
   #Out_Functional_Test.Visual_Test_Approved_PLC_Functional_Test_17 := #_w1 AND #In_Functional_Test.Visual_Test_Approved_PLC_Functional_Test_17;
   IF #_w1 THEN
       #Out_Functional_Test.Electrical_Current_Read_PLC_Functional_Test_17 := #In_Functional_Test.Electrical_Current_Read_PLC_Functional_Test_17;
   END_IF;
   #Out_Functional_Test.Life_Trigger_PLC_Functional_Test_19 := #_w1 AND #In_Functional_Test.Life_Trigger_PLC_Functional_Test_19;
   #Out_Functional_Test.Star_Test_PLC_Functional_Test_19 := #_w1 AND #In_Functional_Test.Star_Test_PLC_Functional_Test_19;
   #Out_Functional_Test.Button_PLC_Functional_Test_19 := #_w1 AND #In_Functional_Test.Button_PLC_Functional_Test_19;
   #Out_Functional_Test.Electrical_Current_Test_Approved_PLC_Functional_Test_19 := #_w1 AND #In_Functional_Test.Electrical_Current_Test_Approved_PLC_Functional_Test_19;
   #Out_Functional_Test.Visual_Test_Approved_PLC_Functional_Test_19 := #_w1 AND #In_Functional_Test.Visual_Test_Approved_PLC_Functional_Test_19;
   IF #_w1 THEN
       #Out_Functional_Test.Electrical_Current_Read_PLC_Functional_Test_19 := #In_Functional_Test.Electrical_Current_Read_PLC_Functional_Test_19;
   END_IF;
   #Out_Functional_Test.Life_Trigger_PLC_Functional_Test_21 := #_w1 AND #In_Functional_Test.Life_Trigger_PLC_Functional_Test_21;
   #Out_Functional_Test.Star_Test_PLC_Functional_Test_21 := #_w1 AND #In_Functional_Test.Star_Test_PLC_Functional_Test_21;
   #Out_Functional_Test.Button_PLC_Functional_Test_21 := #_w1 AND #In_Functional_Test.Button_PLC_Functional_Test_21;
   #Out_Functional_Test.Electrical_Current_Test_Approved_PLC_Functional_Test_21 := #_w1 AND #In_Functional_Test.Electrical_Current_Test_Approved_PLC_Functional_Test_21;
   #Out_Functional_Test.Visual_Test_Approved_PLC_Functional_Test_21 := #_w1 AND #In_Functional_Test.Visual_Test_Approved_PLC_Functional_Test_21;
   IF #_w1 THEN
       #Out_Functional_Test.Electrical_Current_Read_PLC_Functional_Test_21 := #In_Functional_Test.Electrical_Current_Read_PLC_Functional_Test_21;
   END_IF;
   #Out_Functional_Test.Life_Trigger_PLC_Functional_Test_23 := #_w1 AND #In_Functional_Test.Life_Trigger_PLC_Functional_Test_23;
   #Out_Functional_Test.Star_Test_PLC_Functional_Test_23 := #_w1 AND #In_Functional_Test.Star_Test_PLC_Functional_Test_23;
   #Out_Functional_Test.Button_PLC_Functional_Test_23 := #_w1 AND #In_Functional_Test.Button_PLC_Functional_Test_23;
   #Out_Functional_Test.Electrical_Current_Test_Approved_PLC_Functional_Test_23 := #_w1 AND #In_Functional_Test.Electrical_Current_Test_Approved_PLC_Functional_Test_23;
   #Out_Functional_Test.Visual_Test_Approved_PLC_Functional_Test_23 := #_w1 AND #In_Functional_Test.Visual_Test_Approved_PLC_Functional_Test_23;
   IF #_w1 THEN
       #Out_Functional_Test.Electrical_Current_Read_PLC_Functional_Test_23 := #In_Functional_Test.Electrical_Current_Read_PLC_Functional_Test_23;
   END_IF;
   #Out_Functional_Test.Life_Trigger_PLC_Functional_Test_25 := #_w1 AND #In_Functional_Test.Life_Trigger_PLC_Functional_Test_25;
   #Out_Functional_Test.Star_Test_PLC_Functional_Test_25 := #_w1 AND #In_Functional_Test.Star_Test_PLC_Functional_Test_25;
   #Out_Functional_Test.Button_PLC_Functional_Test_25 := #_w1 AND #In_Functional_Test.Button_PLC_Functional_Test_25;
   #Out_Functional_Test.Electrical_Current_Test_Approved_PLC_Functional_Test_25 := #_w1 AND #In_Functional_Test.Electrical_Current_Test_Approved_PLC_Functional_Test_25;
   #Out_Functional_Test.Visual_Test_Approved_PLC_Functional_Test_25 := #_w1 AND #In_Functional_Test.Visual_Test_Approved_PLC_Functional_Test_25;
   IF #_w1 THEN
       #Out_Functional_Test.Electrical_Current_Read_PLC_Functional_Test_25 := #In_Functional_Test.Electrical_Current_Read_PLC_Functional_Test_25;
   END_IF;
   #Out_Functional_Test.Life_Trigger_PLC_Functional_Test_27 := #_w1 AND #In_Functional_Test.Life_Trigger_PLC_Functional_Test_27;
   #Out_Functional_Test.Star_Test_PLC_Functional_Test_27 := #_w1 AND #In_Functional_Test.Star_Test_PLC_Functional_Test_27;
   #Out_Functional_Test.Button_PLC_Functional_Test_27 := #_w1 AND #In_Functional_Test.Button_PLC_Functional_Test_27;
   #Out_Functional_Test.Electrical_Current_Test_Approved_PLC_Functional_Test_27 := #_w1 AND #In_Functional_Test.Electrical_Current_Test_Approved_PLC_Functional_Test_27;
   #Out_Functional_Test.Visual_Test_Approved_PLC_Functional_Test_27 := #_w1 AND #In_Functional_Test.Visual_Test_Approved_PLC_Functional_Test_27;
   IF #_w1 THEN
       #Out_Functional_Test.Electrical_Current_Read_PLC_Functional_Test_27 := #In_Functional_Test.Electrical_Current_Read_PLC_Functional_Test_27;
   END_IF;
   #Out_Functional_Test.Life_Trigger_PLC_Functional_Test_29 := #_w1 AND #In_Functional_Test.Life_Trigger_PLC_Functional_Test_29;
   #Out_Functional_Test.Star_Test_PLC_Functional_Test_29 := #_w1 AND #In_Functional_Test.Star_Test_PLC_Functional_Test_29;
   #Out_Functional_Test.Button_PLC_Functional_Test_29 := #_w1 AND #In_Functional_Test.Button_PLC_Functional_Test_29;
   #Out_Functional_Test.Electrical_Current_Test_Approved_PLC_Functional_Test_29 := #_w1 AND #In_Functional_Test.Electrical_Current_Test_Approved_PLC_Functional_Test_29;
   #Out_Functional_Test.Visual_Test_Approved_PLC_Functional_Test_29 := #_w1 AND #In_Functional_Test.Visual_Test_Approved_PLC_Functional_Test_29;
   IF #_w1 THEN
       #Out_Functional_Test.Electrical_Current_Read_PLC_Functional_Test_29 := #In_Functional_Test.Electrical_Current_Read_PLC_Functional_Test_29;
   END_IF;
END_REGION

REGION Network 3: Functional Test Station 3
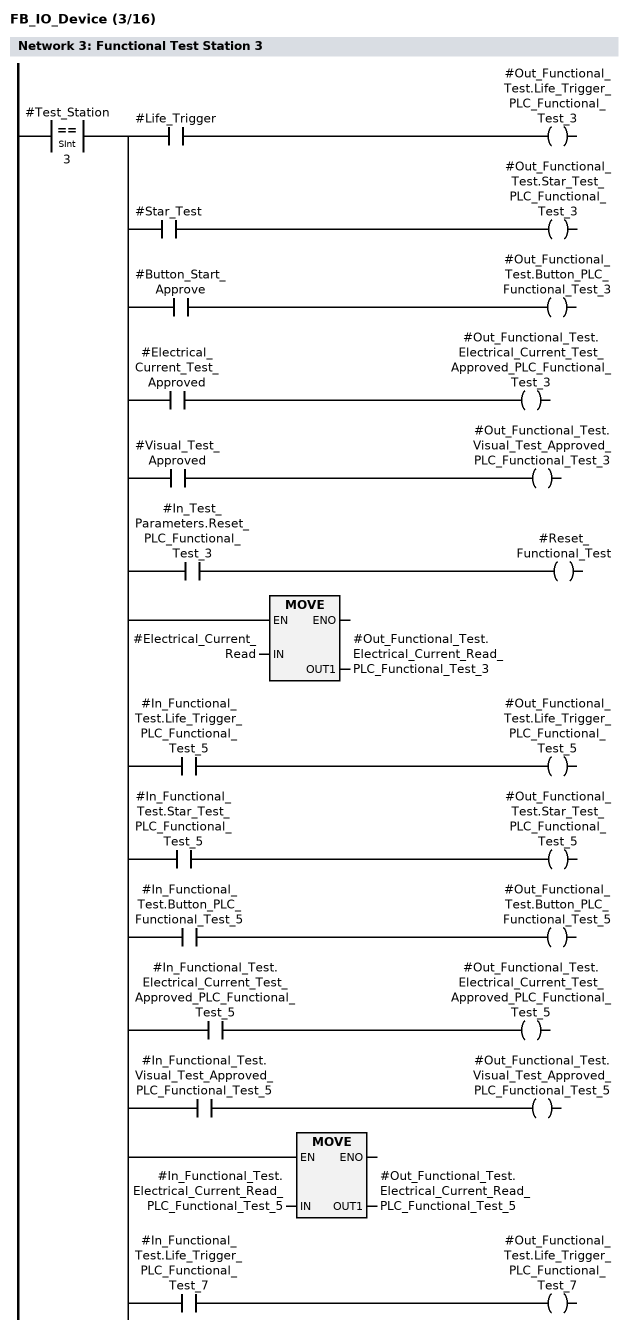
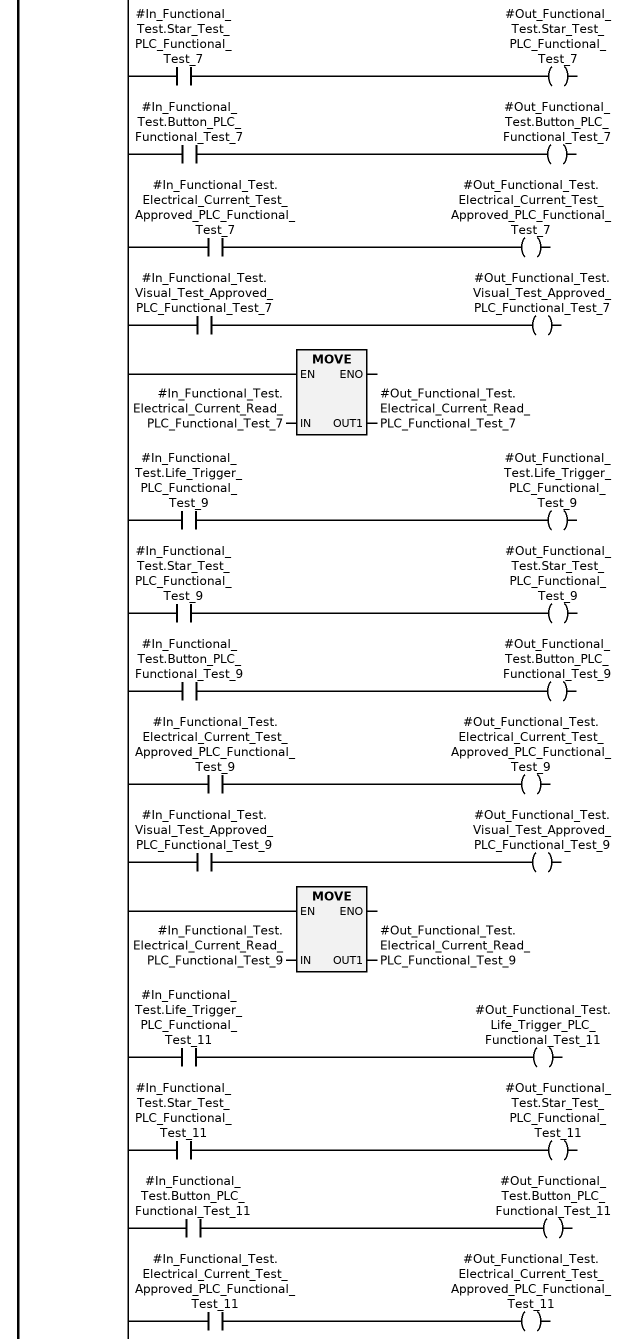
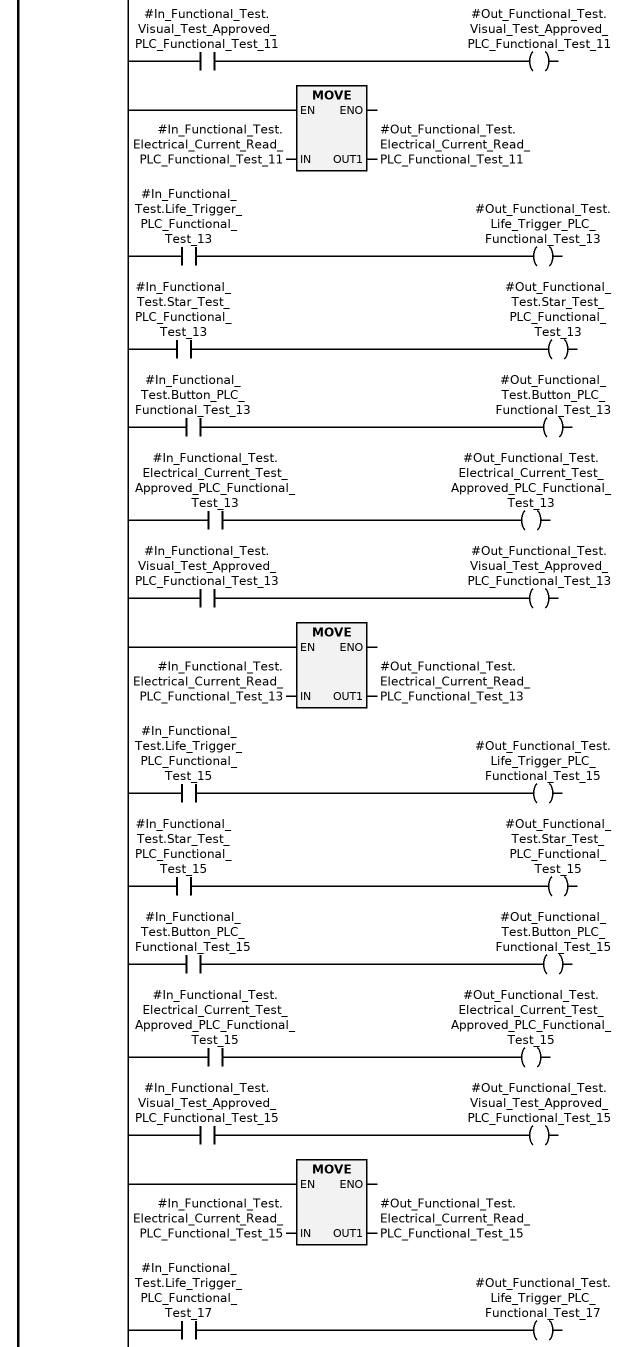
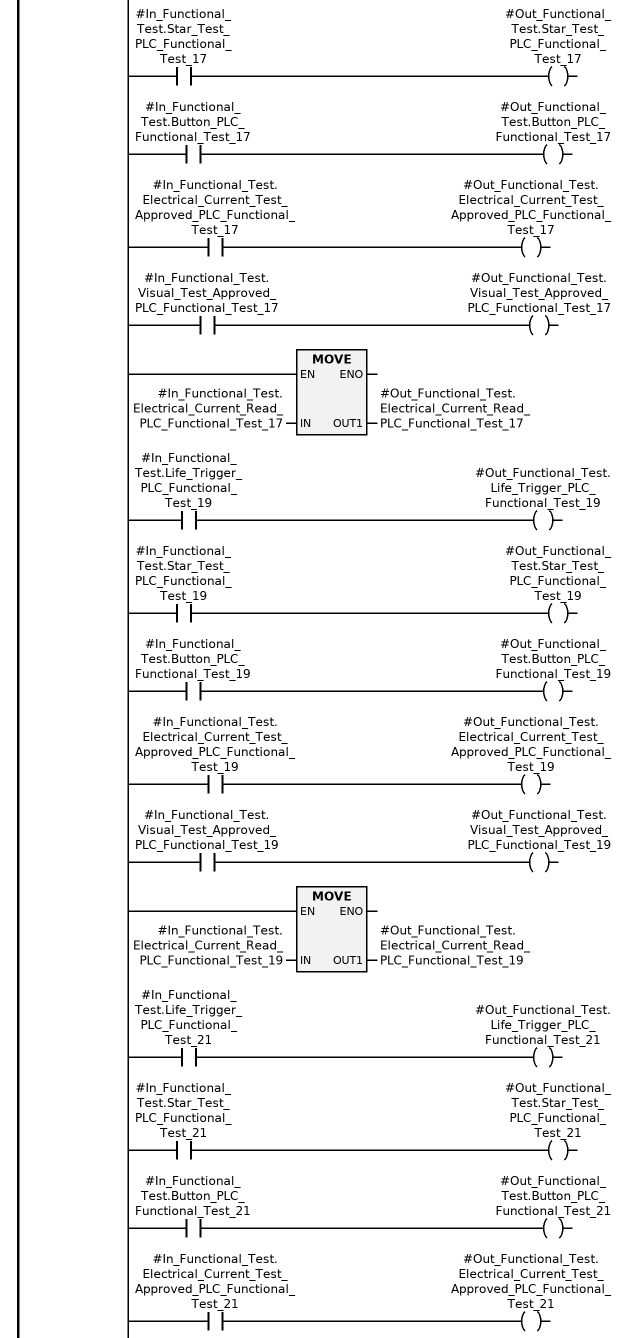
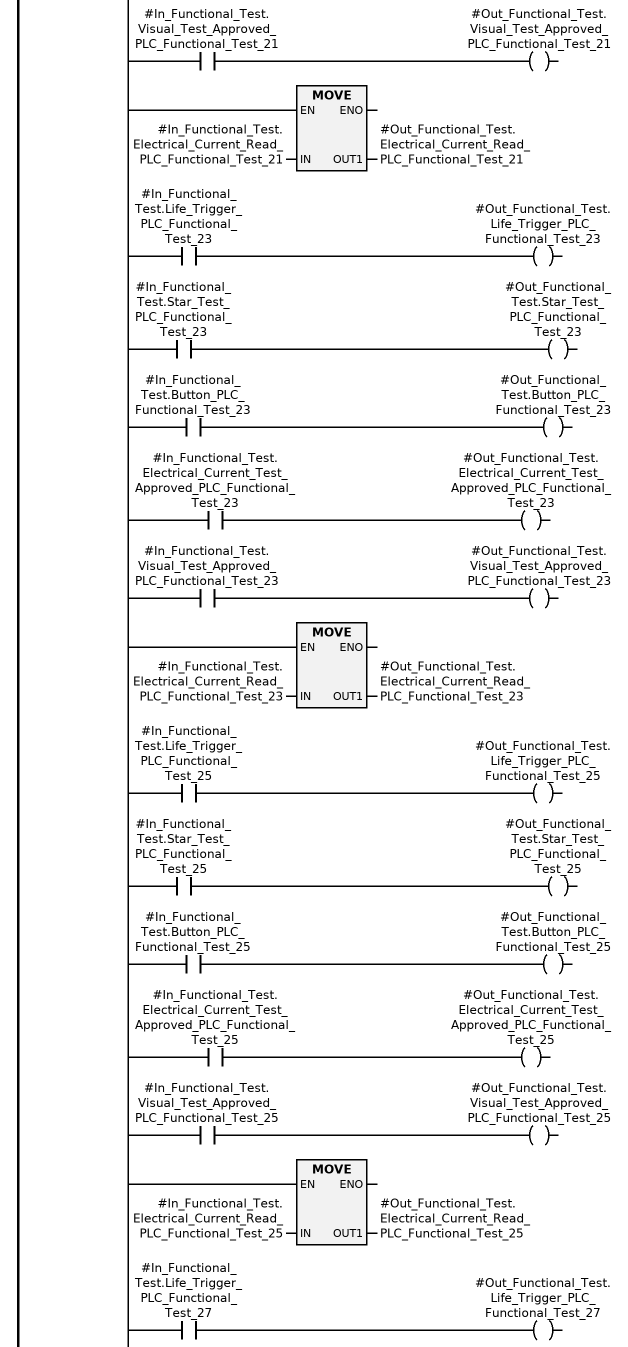
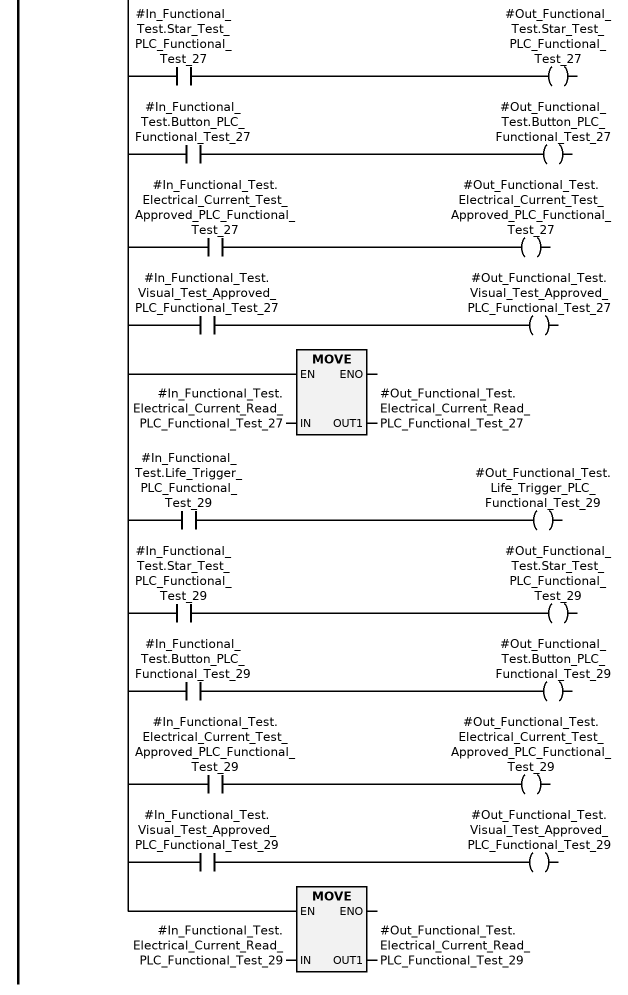
   RUNG wire#powerrail
      { S7_Templates := "SrcType := SInt" } EQ_Contact(in1 := #Test_Station, in2 := 3)
      wire#w1
      Contact( #Life_Trigger )
      Coil( #Out_Functional_Test.Life_Trigger_PLC_Functional_Test_3 )
   END_RUNG
   RUNG wire#w1
      Contact( #Star_Test )
      Coil( #Out_Functional_Test.Star_Test_PLC_Functional_Test_3 )
   END_RUNG
   RUNG wire#w1
      Contact( #Button_Start_Approve )
      Coil( #Out_Functional_Test.Button_PLC_Functional_Test_3 )
   END_RUNG
   RUNG wire#w1
      Contact( #Electrical_Current_Test_Approved )
      Coil( #Out_Functional_Test.Electrical_Current_Test_Approved_PLC_Functional_Test_3 )
   END_RUNG
   RUNG wire#w1
      Contact( #Visual_Test_Approved )
      Coil( #Out_Functional_Test.Visual_Test_Approved_PLC_Functional_Test_3 )
   END_RUNG
   RUNG wire#w1
      Contact( #In_Test_Parameters.Reset_PLC_Functional_Test_3 )
      Coil( #Reset_Functional_Test )
   END_RUNG
   RUNG wire#w1
      Move(in := #Electrical_Current_Read, out1 => #Out_Functional_Test.Electrical_Current_Read_PLC_Functional_Test_3)
   END_RUNG
   RUNG wire#w1
      Contact( #In_Functional_Test.Life_Trigger_PLC_Functional_Test_5 )
      Coil( #Out_Functional_Test.Life_Trigger_PLC_Functional_Test_5 )
   END_RUNG
   RUNG wire#w1
      Contact( #In_Functional_Test.Star_Test_PLC_Functional_Test_5 )
      Coil( #Out_Functional_Test.Star_Test_PLC_Functional_Test_5 )
   END_RUNG
   RUNG wire#w1
      Contact( #In_Functional_Test.Button_PLC_Functional_Test_5 )
      Coil( #Out_Functional_Test.Button_PLC_Functional_Test_5 )
   END_RUNG
   RUNG wire#w1
      Contact( #In_Functional_Test.Electrical_Current_Test_Approved_PLC_Functional_Test_5 )
      Coil( #Out_Functional_Test.Electrical_Current_Test_Approved_PLC_Functional_Test_5 )
   END_RUNG
   RUNG wire#w1
      Contact( #In_Functional_Test.Visual_Test_Approved_PLC_Functional_Test_5 )
      Coil( #Out_Functional_Test.Visual_Test_Approved_PLC_Functional_Test_5 )
   END_RUNG
   RUNG wire#w1
      Move(in := #In_Functional_Test.Electrical_Current_Read_PLC_Functional_Test_5, out1 => #Out_Functional_Test.Electrical_Current_Read_PLC_Functional_Test_5)
   END_RUNG
   RUNG wire#w1
      Contact( #In_Functional_Test.Life_Trigger_PLC_Functional_Test_7 )
      Coil( #Out_Functional_Test.Life_Trigger_PLC_Functional_Test_7 )
   END_RUNG
   RUNG wire#w1
      Contact( #In_Functional_Test.Star_Test_PLC_Functional_Test_7 )
      Coil( #Out_Functional_Test.Star_Test_PLC_Functional_Test_7 )
   END_RUNG
   RUNG wire#w1
      Contact( #In_Functional_Test.Button_PLC_Functional_Test_7 )
      Coil( #Out_Functional_Test.Button_PLC_Functional_Test_7 )
   END_RUNG
   RUNG wire#w1
      Contact( #In_Functional_Test.Electrical_Current_Test_Approved_PLC_Functional_Test_7 )
      Coil( #Out_Functional_Test.Electrical_Current_Test_Approved_PLC_Functional_Test_7 )
   END_RUNG
   RUNG wire#w1
      Contact( #In_Functional_Test.Visual_Test_Approved_PLC_Functional_Test_7 )
      Coil( #Out_Functional_Test.Visual_Test_Approved_PLC_Functional_Test_7 )
   END_RUNG
   RUNG wire#w1
      Move(in := #In_Functional_Test.Electrical_Current_Read_PLC_Functional_Test_7, out1 => #Out_Functional_Test.Electrical_Current_Read_PLC_Functional_Test_7)
   END_RUNG
   RUNG wire#w1
      Contact( #In_Functional_Test.Life_Trigger_PLC_Functional_Test_9 )
      Coil( #Out_Functional_Test.Life_Trigger_PLC_Functional_Test_9 )
   END_RUNG
   RUNG wire#w1
      Contact( #In_Functional_Test.Star_Test_PLC_Functional_Test_9 )
      Coil( #Out_Functional_Test.Star_Test_PLC_Functional_Test_9 )
   END_RUNG
   RUNG wire#w1
      Contact( #In_Functional_Test.Button_PLC_Functional_Test_9 )
      Coil( #Out_Functional_Test.Button_PLC_Functional_Test_9 )
   END_RUNG
   RUNG wire#w1
      Contact( #In_Functional_Test.Electrical_Current_Test_Approved_PLC_Functional_Test_9 )
      Coil( #Out_Functional_Test.Electrical_Current_Test_Approved_PLC_Functional_Test_9 )
   END_RUNG
   RUNG wire#w1
      Contact( #In_Functional_Test.Visual_Test_Approved_PLC_Functional_Test_9 )
      Coil( #Out_Functional_Test.Visual_Test_Approved_PLC_Functional_Test_9 )
   END_RUNG
   RUNG wire#w1
      Move(in := #In_Functional_Test.Electrical_Current_Read_PLC_Functional_Test_9, out1 => #Out_Functional_Test.Electrical_Current_Read_PLC_Functional_Test_9)
   END_RUNG
   RUNG wire#w1
      Contact( #In_Functional_Test.Life_Trigger_PLC_Functional_Test_11 )
      Coil( #Out_Functional_Test.Life_Trigger_PLC_Functional_Test_11 )
   END_RUNG
   RUNG wire#w1
      Contact( #In_Functional_Test.Star_Test_PLC_Functional_Test_11 )
      Coil( #Out_Functional_Test.Star_Test_PLC_Functional_Test_11 )
   END_RUNG
   RUNG wire#w1
      Contact( #In_Functional_Test.Button_PLC_Functional_Test_11 )
      Coil( #Out_Functional_Test.Button_PLC_Functional_Test_11 )
   END_RUNG
   RUNG wire#w1
      Contact( #In_Functional_Test.Electrical_Current_Test_Approved_PLC_Functional_Test_11 )
      Coil( #Out_Functional_Test.Electrical_Current_Test_Approved_PLC_Functional_Test_11 )
   END_RUNG
   RUNG wire#w1
      Contact( #In_Functional_Test.Visual_Test_Approved_PLC_Functional_Test_11 )
      Coil( #Out_Functional_Test.Visual_Test_Approved_PLC_Functional_Test_11 )
   END_RUNG
   RUNG wire#w1
      Move(in := #In_Functional_Test.Electrical_Current_Read_PLC_Functional_Test_11, out1 => #Out_Functional_Test.Electrical_Current_Read_PLC_Functional_Test_11)
   END_RUNG
   RUNG wire#w1
      Contact( #In_Functional_Test.Life_Trigger_PLC_Functional_Test_13 )
      Coil( #Out_Functional_Test.Life_Trigger_PLC_Functional_Test_13 )
   END_RUNG
   RUNG wire#w1
      Contact( #In_Functional_Test.Star_Test_PLC_Functional_Test_13 )
      Coil( #Out_Functional_Test.Star_Test_PLC_Functional_Test_13 )
   END_RUNG
   RUNG wire#w1
      Contact( #In_Functional_Test.Button_PLC_Functional_Test_13 )
      Coil( #Out_Functional_Test.Button_PLC_Functional_Test_13 )
   END_RUNG
   RUNG wire#w1
      Contact( #In_Functional_Test.Electrical_Current_Test_Approved_PLC_Functional_Test_13 )
      Coil( #Out_Functional_Test.Electrical_Current_Test_Approved_PLC_Functional_Test_13 )
   END_RUNG
   RUNG wire#w1
      Contact( #In_Functional_Test.Visual_Test_Approved_PLC_Functional_Test_13 )
      Coil( #Out_Functional_Test.Visual_Test_Approved_PLC_Functional_Test_13 )
   END_RUNG
   RUNG wire#w1
      Move(in := #In_Functional_Test.Electrical_Current_Read_PLC_Functional_Test_13, out1 => #Out_Functional_Test.Electrical_Current_Read_PLC_Functional_Test_13)
   END_RUNG
   RUNG wire#w1
      Contact( #In_Functional_Test.Life_Trigger_PLC_Functional_Test_15 )
      Coil( #Out_Functional_Test.Life_Trigger_PLC_Functional_Test_15 )
   END_RUNG
   RUNG wire#w1
      Contact( #In_Functional_Test.Star_Test_PLC_Functional_Test_15 )
      Coil( #Out_Functional_Test.Star_Test_PLC_Functional_Test_15 )
   END_RUNG
   RUNG wire#w1
      Contact( #In_Functional_Test.Button_PLC_Functional_Test_15 )
      Coil( #Out_Functional_Test.Button_PLC_Functional_Test_15 )
   END_RUNG
   RUNG wire#w1
      Contact( #In_Functional_Test.Electrical_Current_Test_Approved_PLC_Functional_Test_15 )
      Coil( #Out_Functional_Test.Electrical_Current_Test_Approved_PLC_Functional_Test_15 )
   END_RUNG
   RUNG wire#w1
      Contact( #In_Functional_Test.Visual_Test_Approved_PLC_Functional_Test_15 )
      Coil( #Out_Functional_Test.Visual_Test_Approved_PLC_Functional_Test_15 )
   END_RUNG
   RUNG wire#w1
      Move(in := #In_Functional_Test.Electrical_Current_Read_PLC_Functional_Test_15, out1 => #Out_Functional_Test.Electrical_Current_Read_PLC_Functional_Test_15)
   END_RUNG
   RUNG wire#w1
      Contact( #In_Functional_Test.Life_Trigger_PLC_Functional_Test_17 )
      Coil( #Out_Functional_Test.Life_Trigger_PLC_Functional_Test_17 )
   END_RUNG
   RUNG wire#w1
      Contact( #In_Functional_Test.Star_Test_PLC_Functional_Test_17 )
      Coil( #Out_Functional_Test.Star_Test_PLC_Functional_Test_17 )
   END_RUNG
   RUNG wire#w1
      Contact( #In_Functional_Test.Button_PLC_Functional_Test_17 )
      Coil( #Out_Functional_Test.Button_PLC_Functional_Test_17 )
   END_RUNG
   RUNG wire#w1
      Contact( #In_Functional_Test.Electrical_Current_Test_Approved_PLC_Functional_Test_17 )
      Coil( #Out_Functional_Test.Electrical_Current_Test_Approved_PLC_Functional_Test_17 )
   END_RUNG
   RUNG wire#w1
      Contact( #In_Functional_Test.Visual_Test_Approved_PLC_Functional_Test_17 )
      Coil( #Out_Functional_Test.Visual_Test_Approved_PLC_Functional_Test_17 )
   END_RUNG
   RUNG wire#w1
      Move(in := #In_Functional_Test.Electrical_Current_Read_PLC_Functional_Test_17, out1 => #Out_Functional_Test.Electrical_Current_Read_PLC_Functional_Test_17)
   END_RUNG
   RUNG wire#w1
      Contact( #In_Functional_Test.Life_Trigger_PLC_Functional_Test_19 )
      Coil( #Out_Functional_Test.Life_Trigger_PLC_Functional_Test_19 )
   END_RUNG
   RUNG wire#w1
      Contact( #In_Functional_Test.Star_Test_PLC_Functional_Test_19 )
      Coil( #Out_Functional_Test.Star_Test_PLC_Functional_Test_19 )
   END_RUNG
   RUNG wire#w1
      Contact( #In_Functional_Test.Button_PLC_Functional_Test_19 )
      Coil( #Out_Functional_Test.Button_PLC_Functional_Test_19 )
   END_RUNG
   RUNG wire#w1
      Contact( #In_Functional_Test.Electrical_Current_Test_Approved_PLC_Functional_Test_19 )
      Coil( #Out_Functional_Test.Electrical_Current_Test_Approved_PLC_Functional_Test_19 )
   END_RUNG
   RUNG wire#w1
      Contact( #In_Functional_Test.Visual_Test_Approved_PLC_Functional_Test_19 )
      Coil( #Out_Functional_Test.Visual_Test_Approved_PLC_Functional_Test_19 )
   END_RUNG
   RUNG wire#w1
      Move(in := #In_Functional_Test.Electrical_Current_Read_PLC_Functional_Test_19, out1 => #Out_Functional_Test.Electrical_Current_Read_PLC_Functional_Test_19)
   END_RUNG
   RUNG wire#w1
      Contact( #In_Functional_Test.Life_Trigger_PLC_Functional_Test_21 )
      Coil( #Out_Functional_Test.Life_Trigger_PLC_Functional_Test_21 )
   END_RUNG
   RUNG wire#w1
      Contact( #In_Functional_Test.Star_Test_PLC_Functional_Test_21 )
      Coil( #Out_Functional_Test.Star_Test_PLC_Functional_Test_21 )
   END_RUNG
   RUNG wire#w1
      Contact( #In_Functional_Test.Button_PLC_Functional_Test_21 )
      Coil( #Out_Functional_Test.Button_PLC_Functional_Test_21 )
   END_RUNG
   RUNG wire#w1
      Contact( #In_Functional_Test.Electrical_Current_Test_Approved_PLC_Functional_Test_21 )
      Coil( #Out_Functional_Test.Electrical_Current_Test_Approved_PLC_Functional_Test_21 )
   END_RUNG
   RUNG wire#w1
      Contact( #In_Functional_Test.Visual_Test_Approved_PLC_Functional_Test_21 )
      Coil( #Out_Functional_Test.Visual_Test_Approved_PLC_Functional_Test_21 )
   END_RUNG
   RUNG wire#w1
      Move(in := #In_Functional_Test.Electrical_Current_Read_PLC_Functional_Test_21, out1 => #Out_Functional_Test.Electrical_Current_Read_PLC_Functional_Test_21)
   END_RUNG
   RUNG wire#w1
      Contact( #In_Functional_Test.Life_Trigger_PLC_Functional_Test_23 )
      Coil( #Out_Functional_Test.Life_Trigger_PLC_Functional_Test_23 )
   END_RUNG
   RUNG wire#w1
      Contact( #In_Functional_Test.Star_Test_PLC_Functional_Test_23 )
      Coil( #Out_Functional_Test.Star_Test_PLC_Functional_Test_23 )
   END_RUNG
   RUNG wire#w1
      Contact( #In_Functional_Test.Button_PLC_Functional_Test_23 )
      Coil( #Out_Functional_Test.Button_PLC_Functional_Test_23 )
   END_RUNG
   RUNG wire#w1
      Contact( #In_Functional_Test.Electrical_Current_Test_Approved_PLC_Functional_Test_23 )
      Coil( #Out_Functional_Test.Electrical_Current_Test_Approved_PLC_Functional_Test_23 )
   END_RUNG
   RUNG wire#w1
      Contact( #In_Functional_Test.Visual_Test_Approved_PLC_Functional_Test_23 )
      Coil( #Out_Functional_Test.Visual_Test_Approved_PLC_Functional_Test_23 )
   END_RUNG
   RUNG wire#w1
      Move(in := #In_Functional_Test.Electrical_Current_Read_PLC_Functional_Test_23, out1 => #Out_Functional_Test.Electrical_Current_Read_PLC_Functional_Test_23)
   END_RUNG
   RUNG wire#w1
      Contact( #In_Functional_Test.Life_Trigger_PLC_Functional_Test_25 )
      Coil( #Out_Functional_Test.Life_Trigger_PLC_Functional_Test_25 )
   END_RUNG
   RUNG wire#w1
      Contact( #In_Functional_Test.Star_Test_PLC_Functional_Test_25 )
      Coil( #Out_Functional_Test.Star_Test_PLC_Functional_Test_25 )
   END_RUNG
   RUNG wire#w1
      Contact( #In_Functional_Test.Button_PLC_Functional_Test_25 )
      Coil( #Out_Functional_Test.Button_PLC_Functional_Test_25 )
   END_RUNG
   RUNG wire#w1
      Contact( #In_Functional_Test.Electrical_Current_Test_Approved_PLC_Functional_Test_25 )
      Coil( #Out_Functional_Test.Electrical_Current_Test_Approved_PLC_Functional_Test_25 )
   END_RUNG
   RUNG wire#w1
      Contact( #In_Functional_Test.Visual_Test_Approved_PLC_Functional_Test_25 )
      Coil( #Out_Functional_Test.Visual_Test_Approved_PLC_Functional_Test_25 )
   END_RUNG
   RUNG wire#w1
      Move(in := #In_Functional_Test.Electrical_Current_Read_PLC_Functional_Test_25, out1 => #Out_Functional_Test.Electrical_Current_Read_PLC_Functional_Test_25)
   END_RUNG
   RUNG wire#w1
      Contact( #In_Functional_Test.Life_Trigger_PLC_Functional_Test_27 )
      Coil( #Out_Functional_Test.Life_Trigger_PLC_Functional_Test_27 )
   END_RUNG
   RUNG wire#w1
      Contact( #In_Functional_Test.Star_Test_PLC_Functional_Test_27 )
      Coil( #Out_Functional_Test.Star_Test_PLC_Functional_Test_27 )
   END_RUNG
   RUNG wire#w1
      Contact( #In_Functional_Test.Button_PLC_Functional_Test_27 )
      Coil( #Out_Functional_Test.Button_PLC_Functional_Test_27 )
   END_RUNG
   RUNG wire#w1
      Contact( #In_Functional_Test.Electrical_Current_Test_Approved_PLC_Functional_Test_27 )
      Coil( #Out_Functional_Test.Electrical_Current_Test_Approved_PLC_Functional_Test_27 )
   END_RUNG
   RUNG wire#w1
      Contact( #In_Functional_Test.Visual_Test_Approved_PLC_Functional_Test_27 )
      Coil( #Out_Functional_Test.Visual_Test_Approved_PLC_Functional_Test_27 )
   END_RUNG
   RUNG wire#w1
      Move(in := #In_Functional_Test.Electrical_Current_Read_PLC_Functional_Test_27, out1 => #Out_Functional_Test.Electrical_Current_Read_PLC_Functional_Test_27)
   END_RUNG
   RUNG wire#w1
      Contact( #In_Functional_Test.Life_Trigger_PLC_Functional_Test_29 )
      Coil( #Out_Functional_Test.Life_Trigger_PLC_Functional_Test_29 )
   END_RUNG
   RUNG wire#w1
      Contact( #In_Functional_Test.Star_Test_PLC_Functional_Test_29 )
      Coil( #Out_Functional_Test.Star_Test_PLC_Functional_Test_29 )
   END_RUNG
   RUNG wire#w1
      Contact( #In_Functional_Test.Button_PLC_Functional_Test_29 )
      Coil( #Out_Functional_Test.Button_PLC_Functional_Test_29 )
   END_RUNG
   RUNG wire#w1
      Contact( #In_Functional_Test.Electrical_Current_Test_Approved_PLC_Functional_Test_29 )
      Coil( #Out_Functional_Test.Electrical_Current_Test_Approved_PLC_Functional_Test_29 )
   END_RUNG
   RUNG wire#w1
      Contact( #In_Functional_Test.Visual_Test_Approved_PLC_Functional_Test_29 )
      Coil( #Out_Functional_Test.Visual_Test_Approved_PLC_Functional_Test_29 )
   END_RUNG
   RUNG wire#w1
      Move(in := #In_Functional_Test.Electrical_Current_Read_PLC_Functional_Test_29, out1 => #Out_Functional_Test.Electrical_Current_Read_PLC_Functional_Test_29)
   END_RUNG
   // the same network as SCL:
   #_w1 := #Test_Station = 3;
   #Out_Functional_Test.Life_Trigger_PLC_Functional_Test_3 := #_w1 AND #Life_Trigger;
   #Out_Functional_Test.Star_Test_PLC_Functional_Test_3 := #_w1 AND #Star_Test;
   #Out_Functional_Test.Button_PLC_Functional_Test_3 := #_w1 AND #Button_Start_Approve;
   #Out_Functional_Test.Electrical_Current_Test_Approved_PLC_Functional_Test_3 := #_w1 AND #Electrical_Current_Test_Approved;
   #Out_Functional_Test.Visual_Test_Approved_PLC_Functional_Test_3 := #_w1 AND #Visual_Test_Approved;
   #Reset_Functional_Test := #_w1 AND #In_Test_Parameters.Reset_PLC_Functional_Test_3;
   IF #_w1 THEN
       #Out_Functional_Test.Electrical_Current_Read_PLC_Functional_Test_3 := #Electrical_Current_Read;
   END_IF;
   #Out_Functional_Test.Life_Trigger_PLC_Functional_Test_5 := #_w1 AND #In_Functional_Test.Life_Trigger_PLC_Functional_Test_5;
   #Out_Functional_Test.Star_Test_PLC_Functional_Test_5 := #_w1 AND #In_Functional_Test.Star_Test_PLC_Functional_Test_5;
   #Out_Functional_Test.Button_PLC_Functional_Test_5 := #_w1 AND #In_Functional_Test.Button_PLC_Functional_Test_5;
   #Out_Functional_Test.Electrical_Current_Test_Approved_PLC_Functional_Test_5 := #_w1 AND #In_Functional_Test.Electrical_Current_Test_Approved_PLC_Functional_Test_5;
   #Out_Functional_Test.Visual_Test_Approved_PLC_Functional_Test_5 := #_w1 AND #In_Functional_Test.Visual_Test_Approved_PLC_Functional_Test_5;
   IF #_w1 THEN
       #Out_Functional_Test.Electrical_Current_Read_PLC_Functional_Test_5 := #In_Functional_Test.Electrical_Current_Read_PLC_Functional_Test_5;
   END_IF;
   #Out_Functional_Test.Life_Trigger_PLC_Functional_Test_7 := #_w1 AND #In_Functional_Test.Life_Trigger_PLC_Functional_Test_7;
   #Out_Functional_Test.Star_Test_PLC_Functional_Test_7 := #_w1 AND #In_Functional_Test.Star_Test_PLC_Functional_Test_7;
   #Out_Functional_Test.Button_PLC_Functional_Test_7 := #_w1 AND #In_Functional_Test.Button_PLC_Functional_Test_7;
   #Out_Functional_Test.Electrical_Current_Test_Approved_PLC_Functional_Test_7 := #_w1 AND #In_Functional_Test.Electrical_Current_Test_Approved_PLC_Functional_Test_7;
   #Out_Functional_Test.Visual_Test_Approved_PLC_Functional_Test_7 := #_w1 AND #In_Functional_Test.Visual_Test_Approved_PLC_Functional_Test_7;
   IF #_w1 THEN
       #Out_Functional_Test.Electrical_Current_Read_PLC_Functional_Test_7 := #In_Functional_Test.Electrical_Current_Read_PLC_Functional_Test_7;
   END_IF;
   #Out_Functional_Test.Life_Trigger_PLC_Functional_Test_9 := #_w1 AND #In_Functional_Test.Life_Trigger_PLC_Functional_Test_9;
   #Out_Functional_Test.Star_Test_PLC_Functional_Test_9 := #_w1 AND #In_Functional_Test.Star_Test_PLC_Functional_Test_9;
   #Out_Functional_Test.Button_PLC_Functional_Test_9 := #_w1 AND #In_Functional_Test.Button_PLC_Functional_Test_9;
   #Out_Functional_Test.Electrical_Current_Test_Approved_PLC_Functional_Test_9 := #_w1 AND #In_Functional_Test.Electrical_Current_Test_Approved_PLC_Functional_Test_9;
   #Out_Functional_Test.Visual_Test_Approved_PLC_Functional_Test_9 := #_w1 AND #In_Functional_Test.Visual_Test_Approved_PLC_Functional_Test_9;
   IF #_w1 THEN
       #Out_Functional_Test.Electrical_Current_Read_PLC_Functional_Test_9 := #In_Functional_Test.Electrical_Current_Read_PLC_Functional_Test_9;
   END_IF;
   #Out_Functional_Test.Life_Trigger_PLC_Functional_Test_11 := #_w1 AND #In_Functional_Test.Life_Trigger_PLC_Functional_Test_11;
   #Out_Functional_Test.Star_Test_PLC_Functional_Test_11 := #_w1 AND #In_Functional_Test.Star_Test_PLC_Functional_Test_11;
   #Out_Functional_Test.Button_PLC_Functional_Test_11 := #_w1 AND #In_Functional_Test.Button_PLC_Functional_Test_11;
   #Out_Functional_Test.Electrical_Current_Test_Approved_PLC_Functional_Test_11 := #_w1 AND #In_Functional_Test.Electrical_Current_Test_Approved_PLC_Functional_Test_11;
   #Out_Functional_Test.Visual_Test_Approved_PLC_Functional_Test_11 := #_w1 AND #In_Functional_Test.Visual_Test_Approved_PLC_Functional_Test_11;
   IF #_w1 THEN
       #Out_Functional_Test.Electrical_Current_Read_PLC_Functional_Test_11 := #In_Functional_Test.Electrical_Current_Read_PLC_Functional_Test_11;
   END_IF;
   #Out_Functional_Test.Life_Trigger_PLC_Functional_Test_13 := #_w1 AND #In_Functional_Test.Life_Trigger_PLC_Functional_Test_13;
   #Out_Functional_Test.Star_Test_PLC_Functional_Test_13 := #_w1 AND #In_Functional_Test.Star_Test_PLC_Functional_Test_13;
   #Out_Functional_Test.Button_PLC_Functional_Test_13 := #_w1 AND #In_Functional_Test.Button_PLC_Functional_Test_13;
   #Out_Functional_Test.Electrical_Current_Test_Approved_PLC_Functional_Test_13 := #_w1 AND #In_Functional_Test.Electrical_Current_Test_Approved_PLC_Functional_Test_13;
   #Out_Functional_Test.Visual_Test_Approved_PLC_Functional_Test_13 := #_w1 AND #In_Functional_Test.Visual_Test_Approved_PLC_Functional_Test_13;
   IF #_w1 THEN
       #Out_Functional_Test.Electrical_Current_Read_PLC_Functional_Test_13 := #In_Functional_Test.Electrical_Current_Read_PLC_Functional_Test_13;
   END_IF;
   #Out_Functional_Test.Life_Trigger_PLC_Functional_Test_15 := #_w1 AND #In_Functional_Test.Life_Trigger_PLC_Functional_Test_15;
   #Out_Functional_Test.Star_Test_PLC_Functional_Test_15 := #_w1 AND #In_Functional_Test.Star_Test_PLC_Functional_Test_15;
   #Out_Functional_Test.Button_PLC_Functional_Test_15 := #_w1 AND #In_Functional_Test.Button_PLC_Functional_Test_15;
   #Out_Functional_Test.Electrical_Current_Test_Approved_PLC_Functional_Test_15 := #_w1 AND #In_Functional_Test.Electrical_Current_Test_Approved_PLC_Functional_Test_15;
   #Out_Functional_Test.Visual_Test_Approved_PLC_Functional_Test_15 := #_w1 AND #In_Functional_Test.Visual_Test_Approved_PLC_Functional_Test_15;
   IF #_w1 THEN
       #Out_Functional_Test.Electrical_Current_Read_PLC_Functional_Test_15 := #In_Functional_Test.Electrical_Current_Read_PLC_Functional_Test_15;
   END_IF;
   #Out_Functional_Test.Life_Trigger_PLC_Functional_Test_17 := #_w1 AND #In_Functional_Test.Life_Trigger_PLC_Functional_Test_17;
   #Out_Functional_Test.Star_Test_PLC_Functional_Test_17 := #_w1 AND #In_Functional_Test.Star_Test_PLC_Functional_Test_17;
   #Out_Functional_Test.Button_PLC_Functional_Test_17 := #_w1 AND #In_Functional_Test.Button_PLC_Functional_Test_17;
   #Out_Functional_Test.Electrical_Current_Test_Approved_PLC_Functional_Test_17 := #_w1 AND #In_Functional_Test.Electrical_Current_Test_Approved_PLC_Functional_Test_17;
   #Out_Functional_Test.Visual_Test_Approved_PLC_Functional_Test_17 := #_w1 AND #In_Functional_Test.Visual_Test_Approved_PLC_Functional_Test_17;
   IF #_w1 THEN
       #Out_Functional_Test.Electrical_Current_Read_PLC_Functional_Test_17 := #In_Functional_Test.Electrical_Current_Read_PLC_Functional_Test_17;
   END_IF;
   #Out_Functional_Test.Life_Trigger_PLC_Functional_Test_19 := #_w1 AND #In_Functional_Test.Life_Trigger_PLC_Functional_Test_19;
   #Out_Functional_Test.Star_Test_PLC_Functional_Test_19 := #_w1 AND #In_Functional_Test.Star_Test_PLC_Functional_Test_19;
   #Out_Functional_Test.Button_PLC_Functional_Test_19 := #_w1 AND #In_Functional_Test.Button_PLC_Functional_Test_19;
   #Out_Functional_Test.Electrical_Current_Test_Approved_PLC_Functional_Test_19 := #_w1 AND #In_Functional_Test.Electrical_Current_Test_Approved_PLC_Functional_Test_19;
   #Out_Functional_Test.Visual_Test_Approved_PLC_Functional_Test_19 := #_w1 AND #In_Functional_Test.Visual_Test_Approved_PLC_Functional_Test_19;
   IF #_w1 THEN
       #Out_Functional_Test.Electrical_Current_Read_PLC_Functional_Test_19 := #In_Functional_Test.Electrical_Current_Read_PLC_Functional_Test_19;
   END_IF;
   #Out_Functional_Test.Life_Trigger_PLC_Functional_Test_21 := #_w1 AND #In_Functional_Test.Life_Trigger_PLC_Functional_Test_21;
   #Out_Functional_Test.Star_Test_PLC_Functional_Test_21 := #_w1 AND #In_Functional_Test.Star_Test_PLC_Functional_Test_21;
   #Out_Functional_Test.Button_PLC_Functional_Test_21 := #_w1 AND #In_Functional_Test.Button_PLC_Functional_Test_21;
   #Out_Functional_Test.Electrical_Current_Test_Approved_PLC_Functional_Test_21 := #_w1 AND #In_Functional_Test.Electrical_Current_Test_Approved_PLC_Functional_Test_21;
   #Out_Functional_Test.Visual_Test_Approved_PLC_Functional_Test_21 := #_w1 AND #In_Functional_Test.Visual_Test_Approved_PLC_Functional_Test_21;
   IF #_w1 THEN
       #Out_Functional_Test.Electrical_Current_Read_PLC_Functional_Test_21 := #In_Functional_Test.Electrical_Current_Read_PLC_Functional_Test_21;
   END_IF;
   #Out_Functional_Test.Life_Trigger_PLC_Functional_Test_23 := #_w1 AND #In_Functional_Test.Life_Trigger_PLC_Functional_Test_23;
   #Out_Functional_Test.Star_Test_PLC_Functional_Test_23 := #_w1 AND #In_Functional_Test.Star_Test_PLC_Functional_Test_23;
   #Out_Functional_Test.Button_PLC_Functional_Test_23 := #_w1 AND #In_Functional_Test.Button_PLC_Functional_Test_23;
   #Out_Functional_Test.Electrical_Current_Test_Approved_PLC_Functional_Test_23 := #_w1 AND #In_Functional_Test.Electrical_Current_Test_Approved_PLC_Functional_Test_23;
   #Out_Functional_Test.Visual_Test_Approved_PLC_Functional_Test_23 := #_w1 AND #In_Functional_Test.Visual_Test_Approved_PLC_Functional_Test_23;
   IF #_w1 THEN
       #Out_Functional_Test.Electrical_Current_Read_PLC_Functional_Test_23 := #In_Functional_Test.Electrical_Current_Read_PLC_Functional_Test_23;
   END_IF;
   #Out_Functional_Test.Life_Trigger_PLC_Functional_Test_25 := #_w1 AND #In_Functional_Test.Life_Trigger_PLC_Functional_Test_25;
   #Out_Functional_Test.Star_Test_PLC_Functional_Test_25 := #_w1 AND #In_Functional_Test.Star_Test_PLC_Functional_Test_25;
   #Out_Functional_Test.Button_PLC_Functional_Test_25 := #_w1 AND #In_Functional_Test.Button_PLC_Functional_Test_25;
   #Out_Functional_Test.Electrical_Current_Test_Approved_PLC_Functional_Test_25 := #_w1 AND #In_Functional_Test.Electrical_Current_Test_Approved_PLC_Functional_Test_25;
   #Out_Functional_Test.Visual_Test_Approved_PLC_Functional_Test_25 := #_w1 AND #In_Functional_Test.Visual_Test_Approved_PLC_Functional_Test_25;
   IF #_w1 THEN
       #Out_Functional_Test.Electrical_Current_Read_PLC_Functional_Test_25 := #In_Functional_Test.Electrical_Current_Read_PLC_Functional_Test_25;
   END_IF;
   #Out_Functional_Test.Life_Trigger_PLC_Functional_Test_27 := #_w1 AND #In_Functional_Test.Life_Trigger_PLC_Functional_Test_27;
   #Out_Functional_Test.Star_Test_PLC_Functional_Test_27 := #_w1 AND #In_Functional_Test.Star_Test_PLC_Functional_Test_27;
   #Out_Functional_Test.Button_PLC_Functional_Test_27 := #_w1 AND #In_Functional_Test.Button_PLC_Functional_Test_27;
   #Out_Functional_Test.Electrical_Current_Test_Approved_PLC_Functional_Test_27 := #_w1 AND #In_Functional_Test.Electrical_Current_Test_Approved_PLC_Functional_Test_27;
   #Out_Functional_Test.Visual_Test_Approved_PLC_Functional_Test_27 := #_w1 AND #In_Functional_Test.Visual_Test_Approved_PLC_Functional_Test_27;
   IF #_w1 THEN
       #Out_Functional_Test.Electrical_Current_Read_PLC_Functional_Test_27 := #In_Functional_Test.Electrical_Current_Read_PLC_Functional_Test_27;
   END_IF;
   #Out_Functional_Test.Life_Trigger_PLC_Functional_Test_29 := #_w1 AND #In_Functional_Test.Life_Trigger_PLC_Functional_Test_29;
   #Out_Functional_Test.Star_Test_PLC_Functional_Test_29 := #_w1 AND #In_Functional_Test.Star_Test_PLC_Functional_Test_29;
   #Out_Functional_Test.Button_PLC_Functional_Test_29 := #_w1 AND #In_Functional_Test.Button_PLC_Functional_Test_29;
   #Out_Functional_Test.Electrical_Current_Test_Approved_PLC_Functional_Test_29 := #_w1 AND #In_Functional_Test.Electrical_Current_Test_Approved_PLC_Functional_Test_29;
   #Out_Functional_Test.Visual_Test_Approved_PLC_Functional_Test_29 := #_w1 AND #In_Functional_Test.Visual_Test_Approved_PLC_Functional_Test_29;
   IF #_w1 THEN
       #Out_Functional_Test.Electrical_Current_Read_PLC_Functional_Test_29 := #In_Functional_Test.Electrical_Current_Read_PLC_Functional_Test_29;
   END_IF;
END_REGION

REGION Network 4: Functional Test Station 5
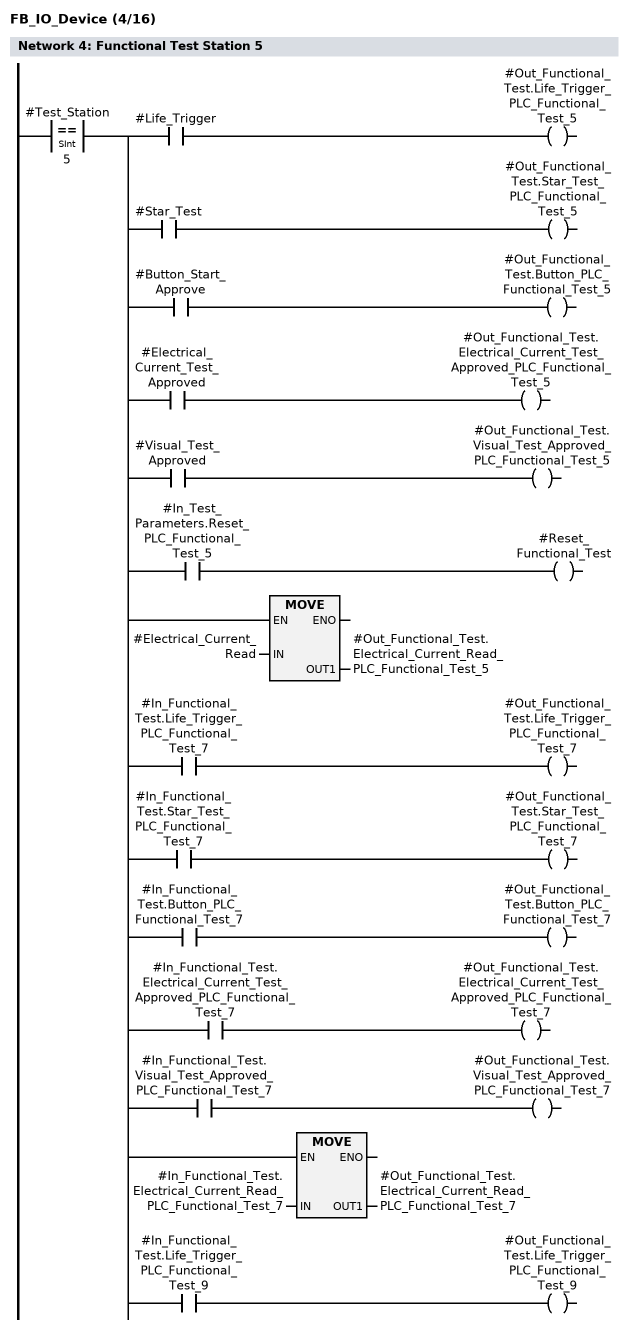
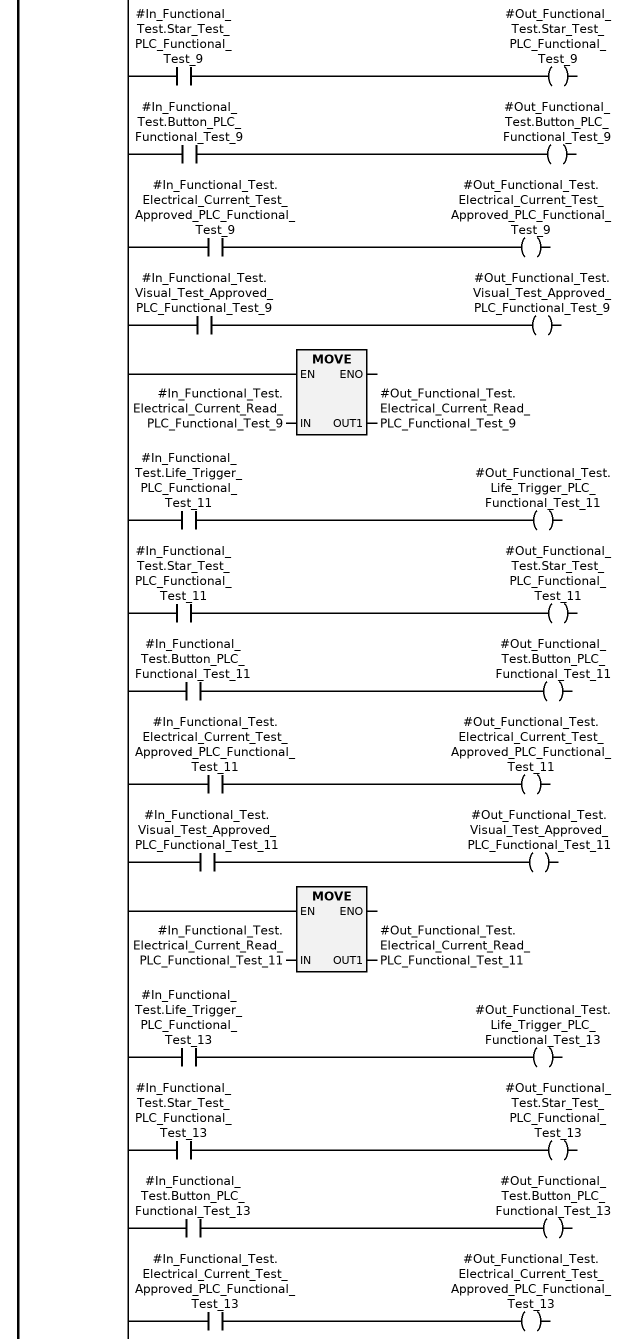
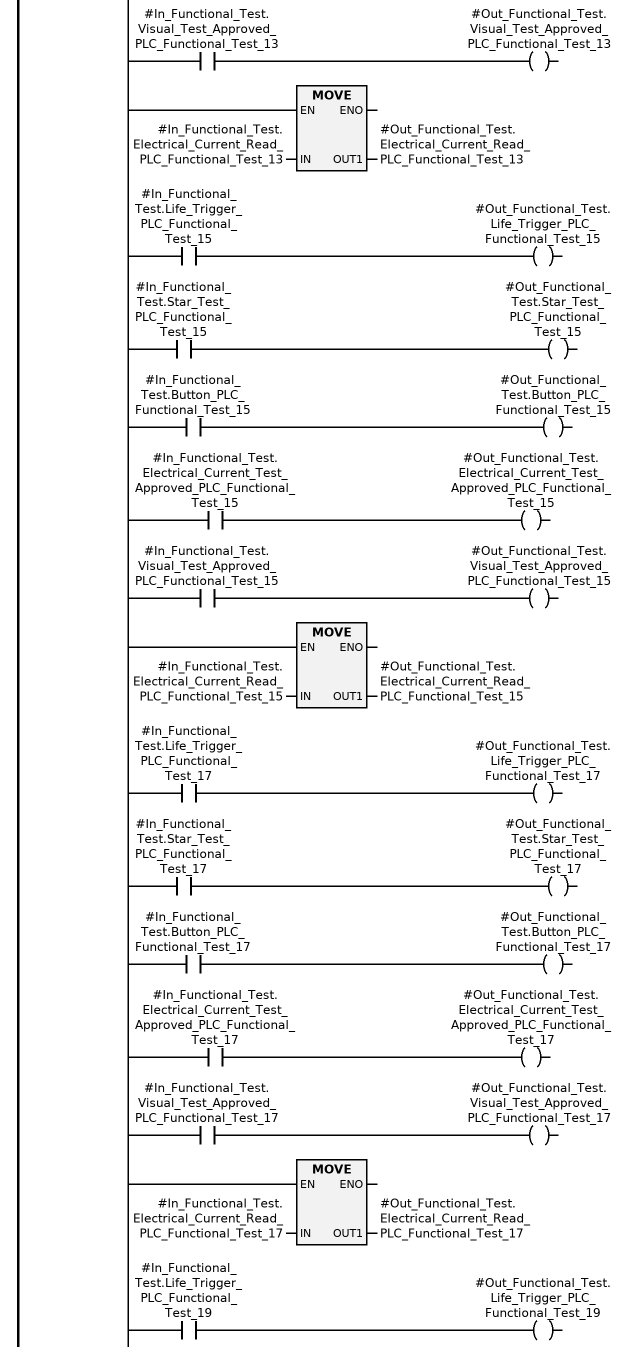
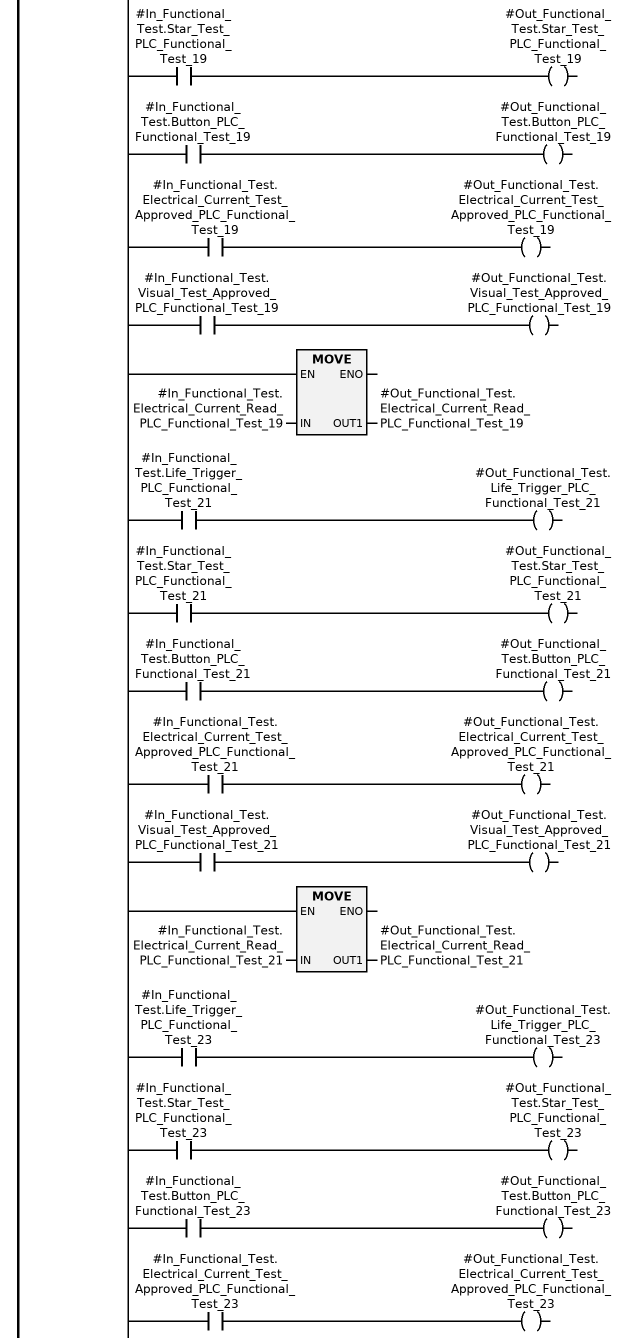
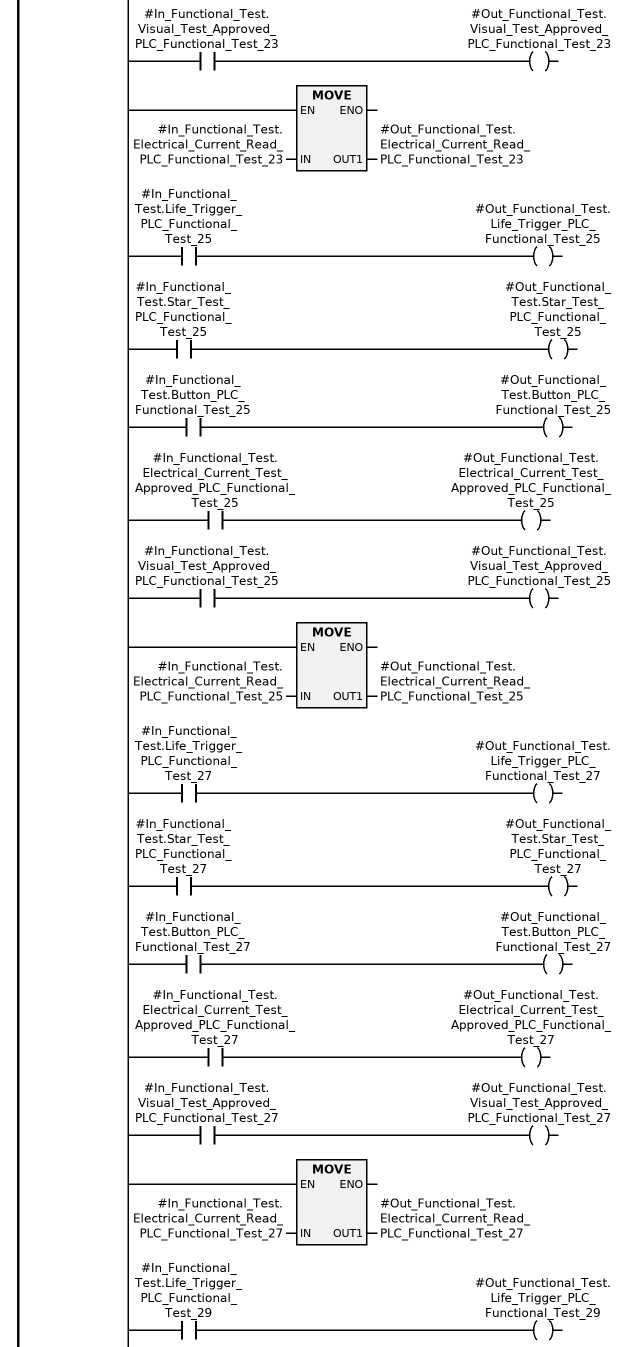
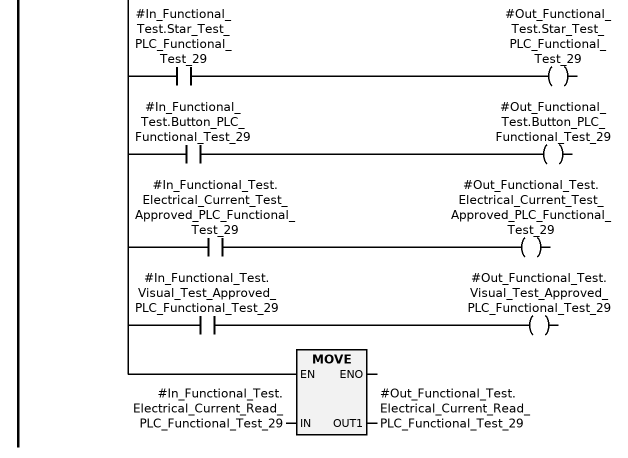
   RUNG wire#powerrail
      { S7_Templates := "SrcType := SInt" } EQ_Contact(in1 := #Test_Station, in2 := 5)
      wire#w1
      Contact( #Life_Trigger )
      Coil( #Out_Functional_Test.Life_Trigger_PLC_Functional_Test_5 )
   END_RUNG
   RUNG wire#w1
      Contact( #Star_Test )
      Coil( #Out_Functional_Test.Star_Test_PLC_Functional_Test_5 )
   END_RUNG
   RUNG wire#w1
      Contact( #Button_Start_Approve )
      Coil( #Out_Functional_Test.Button_PLC_Functional_Test_5 )
   END_RUNG
   RUNG wire#w1
      Contact( #Electrical_Current_Test_Approved )
      Coil( #Out_Functional_Test.Electrical_Current_Test_Approved_PLC_Functional_Test_5 )
   END_RUNG
   RUNG wire#w1
      Contact( #Visual_Test_Approved )
      Coil( #Out_Functional_Test.Visual_Test_Approved_PLC_Functional_Test_5 )
   END_RUNG
   RUNG wire#w1
      Contact( #In_Test_Parameters.Reset_PLC_Functional_Test_5 )
      Coil( #Reset_Functional_Test )
   END_RUNG
   RUNG wire#w1
      Move(in := #Electrical_Current_Read, out1 => #Out_Functional_Test.Electrical_Current_Read_PLC_Functional_Test_5)
   END_RUNG
   RUNG wire#w1
      Contact( #In_Functional_Test.Life_Trigger_PLC_Functional_Test_7 )
      Coil( #Out_Functional_Test.Life_Trigger_PLC_Functional_Test_7 )
   END_RUNG
   RUNG wire#w1
      Contact( #In_Functional_Test.Star_Test_PLC_Functional_Test_7 )
      Coil( #Out_Functional_Test.Star_Test_PLC_Functional_Test_7 )
   END_RUNG
   RUNG wire#w1
      Contact( #In_Functional_Test.Button_PLC_Functional_Test_7 )
      Coil( #Out_Functional_Test.Button_PLC_Functional_Test_7 )
   END_RUNG
   RUNG wire#w1
      Contact( #In_Functional_Test.Electrical_Current_Test_Approved_PLC_Functional_Test_7 )
      Coil( #Out_Functional_Test.Electrical_Current_Test_Approved_PLC_Functional_Test_7 )
   END_RUNG
   RUNG wire#w1
      Contact( #In_Functional_Test.Visual_Test_Approved_PLC_Functional_Test_7 )
      Coil( #Out_Functional_Test.Visual_Test_Approved_PLC_Functional_Test_7 )
   END_RUNG
   RUNG wire#w1
      Move(in := #In_Functional_Test.Electrical_Current_Read_PLC_Functional_Test_7, out1 => #Out_Functional_Test.Electrical_Current_Read_PLC_Functional_Test_7)
   END_RUNG
   RUNG wire#w1
      Contact( #In_Functional_Test.Life_Trigger_PLC_Functional_Test_9 )
      Coil( #Out_Functional_Test.Life_Trigger_PLC_Functional_Test_9 )
   END_RUNG
   RUNG wire#w1
      Contact( #In_Functional_Test.Star_Test_PLC_Functional_Test_9 )
      Coil( #Out_Functional_Test.Star_Test_PLC_Functional_Test_9 )
   END_RUNG
   RUNG wire#w1
      Contact( #In_Functional_Test.Button_PLC_Functional_Test_9 )
      Coil( #Out_Functional_Test.Button_PLC_Functional_Test_9 )
   END_RUNG
   RUNG wire#w1
      Contact( #In_Functional_Test.Electrical_Current_Test_Approved_PLC_Functional_Test_9 )
      Coil( #Out_Functional_Test.Electrical_Current_Test_Approved_PLC_Functional_Test_9 )
   END_RUNG
   RUNG wire#w1
      Contact( #In_Functional_Test.Visual_Test_Approved_PLC_Functional_Test_9 )
      Coil( #Out_Functional_Test.Visual_Test_Approved_PLC_Functional_Test_9 )
   END_RUNG
   RUNG wire#w1
      Move(in := #In_Functional_Test.Electrical_Current_Read_PLC_Functional_Test_9, out1 => #Out_Functional_Test.Electrical_Current_Read_PLC_Functional_Test_9)
   END_RUNG
   RUNG wire#w1
      Contact( #In_Functional_Test.Life_Trigger_PLC_Functional_Test_11 )
      Coil( #Out_Functional_Test.Life_Trigger_PLC_Functional_Test_11 )
   END_RUNG
   RUNG wire#w1
      Contact( #In_Functional_Test.Star_Test_PLC_Functional_Test_11 )
      Coil( #Out_Functional_Test.Star_Test_PLC_Functional_Test_11 )
   END_RUNG
   RUNG wire#w1
      Contact( #In_Functional_Test.Button_PLC_Functional_Test_11 )
      Coil( #Out_Functional_Test.Button_PLC_Functional_Test_11 )
   END_RUNG
   RUNG wire#w1
      Contact( #In_Functional_Test.Electrical_Current_Test_Approved_PLC_Functional_Test_11 )
      Coil( #Out_Functional_Test.Electrical_Current_Test_Approved_PLC_Functional_Test_11 )
   END_RUNG
   RUNG wire#w1
      Contact( #In_Functional_Test.Visual_Test_Approved_PLC_Functional_Test_11 )
      Coil( #Out_Functional_Test.Visual_Test_Approved_PLC_Functional_Test_11 )
   END_RUNG
   RUNG wire#w1
      Move(in := #In_Functional_Test.Electrical_Current_Read_PLC_Functional_Test_11, out1 => #Out_Functional_Test.Electrical_Current_Read_PLC_Functional_Test_11)
   END_RUNG
   RUNG wire#w1
      Contact( #In_Functional_Test.Life_Trigger_PLC_Functional_Test_13 )
      Coil( #Out_Functional_Test.Life_Trigger_PLC_Functional_Test_13 )
   END_RUNG
   RUNG wire#w1
      Contact( #In_Functional_Test.Star_Test_PLC_Functional_Test_13 )
      Coil( #Out_Functional_Test.Star_Test_PLC_Functional_Test_13 )
   END_RUNG
   RUNG wire#w1
      Contact( #In_Functional_Test.Button_PLC_Functional_Test_13 )
      Coil( #Out_Functional_Test.Button_PLC_Functional_Test_13 )
   END_RUNG
   RUNG wire#w1
      Contact( #In_Functional_Test.Electrical_Current_Test_Approved_PLC_Functional_Test_13 )
      Coil( #Out_Functional_Test.Electrical_Current_Test_Approved_PLC_Functional_Test_13 )
   END_RUNG
   RUNG wire#w1
      Contact( #In_Functional_Test.Visual_Test_Approved_PLC_Functional_Test_13 )
      Coil( #Out_Functional_Test.Visual_Test_Approved_PLC_Functional_Test_13 )
   END_RUNG
   RUNG wire#w1
      Move(in := #In_Functional_Test.Electrical_Current_Read_PLC_Functional_Test_13, out1 => #Out_Functional_Test.Electrical_Current_Read_PLC_Functional_Test_13)
   END_RUNG
   RUNG wire#w1
      Contact( #In_Functional_Test.Life_Trigger_PLC_Functional_Test_15 )
      Coil( #Out_Functional_Test.Life_Trigger_PLC_Functional_Test_15 )
   END_RUNG
   RUNG wire#w1
      Contact( #In_Functional_Test.Star_Test_PLC_Functional_Test_15 )
      Coil( #Out_Functional_Test.Star_Test_PLC_Functional_Test_15 )
   END_RUNG
   RUNG wire#w1
      Contact( #In_Functional_Test.Button_PLC_Functional_Test_15 )
      Coil( #Out_Functional_Test.Button_PLC_Functional_Test_15 )
   END_RUNG
   RUNG wire#w1
      Contact( #In_Functional_Test.Electrical_Current_Test_Approved_PLC_Functional_Test_15 )
      Coil( #Out_Functional_Test.Electrical_Current_Test_Approved_PLC_Functional_Test_15 )
   END_RUNG
   RUNG wire#w1
      Contact( #In_Functional_Test.Visual_Test_Approved_PLC_Functional_Test_15 )
      Coil( #Out_Functional_Test.Visual_Test_Approved_PLC_Functional_Test_15 )
   END_RUNG
   RUNG wire#w1
      Move(in := #In_Functional_Test.Electrical_Current_Read_PLC_Functional_Test_15, out1 => #Out_Functional_Test.Electrical_Current_Read_PLC_Functional_Test_15)
   END_RUNG
   RUNG wire#w1
      Contact( #In_Functional_Test.Life_Trigger_PLC_Functional_Test_17 )
      Coil( #Out_Functional_Test.Life_Trigger_PLC_Functional_Test_17 )
   END_RUNG
   RUNG wire#w1
      Contact( #In_Functional_Test.Star_Test_PLC_Functional_Test_17 )
      Coil( #Out_Functional_Test.Star_Test_PLC_Functional_Test_17 )
   END_RUNG
   RUNG wire#w1
      Contact( #In_Functional_Test.Button_PLC_Functional_Test_17 )
      Coil( #Out_Functional_Test.Button_PLC_Functional_Test_17 )
   END_RUNG
   RUNG wire#w1
      Contact( #In_Functional_Test.Electrical_Current_Test_Approved_PLC_Functional_Test_17 )
      Coil( #Out_Functional_Test.Electrical_Current_Test_Approved_PLC_Functional_Test_17 )
   END_RUNG
   RUNG wire#w1
      Contact( #In_Functional_Test.Visual_Test_Approved_PLC_Functional_Test_17 )
      Coil( #Out_Functional_Test.Visual_Test_Approved_PLC_Functional_Test_17 )
   END_RUNG
   RUNG wire#w1
      Move(in := #In_Functional_Test.Electrical_Current_Read_PLC_Functional_Test_17, out1 => #Out_Functional_Test.Electrical_Current_Read_PLC_Functional_Test_17)
   END_RUNG
   RUNG wire#w1
      Contact( #In_Functional_Test.Life_Trigger_PLC_Functional_Test_19 )
      Coil( #Out_Functional_Test.Life_Trigger_PLC_Functional_Test_19 )
   END_RUNG
   RUNG wire#w1
      Contact( #In_Functional_Test.Star_Test_PLC_Functional_Test_19 )
      Coil( #Out_Functional_Test.Star_Test_PLC_Functional_Test_19 )
   END_RUNG
   RUNG wire#w1
      Contact( #In_Functional_Test.Button_PLC_Functional_Test_19 )
      Coil( #Out_Functional_Test.Button_PLC_Functional_Test_19 )
   END_RUNG
   RUNG wire#w1
      Contact( #In_Functional_Test.Electrical_Current_Test_Approved_PLC_Functional_Test_19 )
      Coil( #Out_Functional_Test.Electrical_Current_Test_Approved_PLC_Functional_Test_19 )
   END_RUNG
   RUNG wire#w1
      Contact( #In_Functional_Test.Visual_Test_Approved_PLC_Functional_Test_19 )
      Coil( #Out_Functional_Test.Visual_Test_Approved_PLC_Functional_Test_19 )
   END_RUNG
   RUNG wire#w1
      Move(in := #In_Functional_Test.Electrical_Current_Read_PLC_Functional_Test_19, out1 => #Out_Functional_Test.Electrical_Current_Read_PLC_Functional_Test_19)
   END_RUNG
   RUNG wire#w1
      Contact( #In_Functional_Test.Life_Trigger_PLC_Functional_Test_21 )
      Coil( #Out_Functional_Test.Life_Trigger_PLC_Functional_Test_21 )
   END_RUNG
   RUNG wire#w1
      Contact( #In_Functional_Test.Star_Test_PLC_Functional_Test_21 )
      Coil( #Out_Functional_Test.Star_Test_PLC_Functional_Test_21 )
   END_RUNG
   RUNG wire#w1
      Contact( #In_Functional_Test.Button_PLC_Functional_Test_21 )
      Coil( #Out_Functional_Test.Button_PLC_Functional_Test_21 )
   END_RUNG
   RUNG wire#w1
      Contact( #In_Functional_Test.Electrical_Current_Test_Approved_PLC_Functional_Test_21 )
      Coil( #Out_Functional_Test.Electrical_Current_Test_Approved_PLC_Functional_Test_21 )
   END_RUNG
   RUNG wire#w1
      Contact( #In_Functional_Test.Visual_Test_Approved_PLC_Functional_Test_21 )
      Coil( #Out_Functional_Test.Visual_Test_Approved_PLC_Functional_Test_21 )
   END_RUNG
   RUNG wire#w1
      Move(in := #In_Functional_Test.Electrical_Current_Read_PLC_Functional_Test_21, out1 => #Out_Functional_Test.Electrical_Current_Read_PLC_Functional_Test_21)
   END_RUNG
   RUNG wire#w1
      Contact( #In_Functional_Test.Life_Trigger_PLC_Functional_Test_23 )
      Coil( #Out_Functional_Test.Life_Trigger_PLC_Functional_Test_23 )
   END_RUNG
   RUNG wire#w1
      Contact( #In_Functional_Test.Star_Test_PLC_Functional_Test_23 )
      Coil( #Out_Functional_Test.Star_Test_PLC_Functional_Test_23 )
   END_RUNG
   RUNG wire#w1
      Contact( #In_Functional_Test.Button_PLC_Functional_Test_23 )
      Coil( #Out_Functional_Test.Button_PLC_Functional_Test_23 )
   END_RUNG
   RUNG wire#w1
      Contact( #In_Functional_Test.Electrical_Current_Test_Approved_PLC_Functional_Test_23 )
      Coil( #Out_Functional_Test.Electrical_Current_Test_Approved_PLC_Functional_Test_23 )
   END_RUNG
   RUNG wire#w1
      Contact( #In_Functional_Test.Visual_Test_Approved_PLC_Functional_Test_23 )
      Coil( #Out_Functional_Test.Visual_Test_Approved_PLC_Functional_Test_23 )
   END_RUNG
   RUNG wire#w1
      Move(in := #In_Functional_Test.Electrical_Current_Read_PLC_Functional_Test_23, out1 => #Out_Functional_Test.Electrical_Current_Read_PLC_Functional_Test_23)
   END_RUNG
   RUNG wire#w1
      Contact( #In_Functional_Test.Life_Trigger_PLC_Functional_Test_25 )
      Coil( #Out_Functional_Test.Life_Trigger_PLC_Functional_Test_25 )
   END_RUNG
   RUNG wire#w1
      Contact( #In_Functional_Test.Star_Test_PLC_Functional_Test_25 )
      Coil( #Out_Functional_Test.Star_Test_PLC_Functional_Test_25 )
   END_RUNG
   RUNG wire#w1
      Contact( #In_Functional_Test.Button_PLC_Functional_Test_25 )
      Coil( #Out_Functional_Test.Button_PLC_Functional_Test_25 )
   END_RUNG
   RUNG wire#w1
      Contact( #In_Functional_Test.Electrical_Current_Test_Approved_PLC_Functional_Test_25 )
      Coil( #Out_Functional_Test.Electrical_Current_Test_Approved_PLC_Functional_Test_25 )
   END_RUNG
   RUNG wire#w1
      Contact( #In_Functional_Test.Visual_Test_Approved_PLC_Functional_Test_25 )
      Coil( #Out_Functional_Test.Visual_Test_Approved_PLC_Functional_Test_25 )
   END_RUNG
   RUNG wire#w1
      Move(in := #In_Functional_Test.Electrical_Current_Read_PLC_Functional_Test_25, out1 => #Out_Functional_Test.Electrical_Current_Read_PLC_Functional_Test_25)
   END_RUNG
   RUNG wire#w1
      Contact( #In_Functional_Test.Life_Trigger_PLC_Functional_Test_27 )
      Coil( #Out_Functional_Test.Life_Trigger_PLC_Functional_Test_27 )
   END_RUNG
   RUNG wire#w1
      Contact( #In_Functional_Test.Star_Test_PLC_Functional_Test_27 )
      Coil( #Out_Functional_Test.Star_Test_PLC_Functional_Test_27 )
   END_RUNG
   RUNG wire#w1
      Contact( #In_Functional_Test.Button_PLC_Functional_Test_27 )
      Coil( #Out_Functional_Test.Button_PLC_Functional_Test_27 )
   END_RUNG
   RUNG wire#w1
      Contact( #In_Functional_Test.Electrical_Current_Test_Approved_PLC_Functional_Test_27 )
      Coil( #Out_Functional_Test.Electrical_Current_Test_Approved_PLC_Functional_Test_27 )
   END_RUNG
   RUNG wire#w1
      Contact( #In_Functional_Test.Visual_Test_Approved_PLC_Functional_Test_27 )
      Coil( #Out_Functional_Test.Visual_Test_Approved_PLC_Functional_Test_27 )
   END_RUNG
   RUNG wire#w1
      Move(in := #In_Functional_Test.Electrical_Current_Read_PLC_Functional_Test_27, out1 => #Out_Functional_Test.Electrical_Current_Read_PLC_Functional_Test_27)
   END_RUNG
   RUNG wire#w1
      Contact( #In_Functional_Test.Life_Trigger_PLC_Functional_Test_29 )
      Coil( #Out_Functional_Test.Life_Trigger_PLC_Functional_Test_29 )
   END_RUNG
   RUNG wire#w1
      Contact( #In_Functional_Test.Star_Test_PLC_Functional_Test_29 )
      Coil( #Out_Functional_Test.Star_Test_PLC_Functional_Test_29 )
   END_RUNG
   RUNG wire#w1
      Contact( #In_Functional_Test.Button_PLC_Functional_Test_29 )
      Coil( #Out_Functional_Test.Button_PLC_Functional_Test_29 )
   END_RUNG
   RUNG wire#w1
      Contact( #In_Functional_Test.Electrical_Current_Test_Approved_PLC_Functional_Test_29 )
      Coil( #Out_Functional_Test.Electrical_Current_Test_Approved_PLC_Functional_Test_29 )
   END_RUNG
   RUNG wire#w1
      Contact( #In_Functional_Test.Visual_Test_Approved_PLC_Functional_Test_29 )
      Coil( #Out_Functional_Test.Visual_Test_Approved_PLC_Functional_Test_29 )
   END_RUNG
   RUNG wire#w1
      Move(in := #In_Functional_Test.Electrical_Current_Read_PLC_Functional_Test_29, out1 => #Out_Functional_Test.Electrical_Current_Read_PLC_Functional_Test_29)
   END_RUNG
   // the same network as SCL:
   #_w1 := #Test_Station = 5;
   #Out_Functional_Test.Life_Trigger_PLC_Functional_Test_5 := #_w1 AND #Life_Trigger;
   #Out_Functional_Test.Star_Test_PLC_Functional_Test_5 := #_w1 AND #Star_Test;
   #Out_Functional_Test.Button_PLC_Functional_Test_5 := #_w1 AND #Button_Start_Approve;
   #Out_Functional_Test.Electrical_Current_Test_Approved_PLC_Functional_Test_5 := #_w1 AND #Electrical_Current_Test_Approved;
   #Out_Functional_Test.Visual_Test_Approved_PLC_Functional_Test_5 := #_w1 AND #Visual_Test_Approved;
   #Reset_Functional_Test := #_w1 AND #In_Test_Parameters.Reset_PLC_Functional_Test_5;
   IF #_w1 THEN
       #Out_Functional_Test.Electrical_Current_Read_PLC_Functional_Test_5 := #Electrical_Current_Read;
   END_IF;
   #Out_Functional_Test.Life_Trigger_PLC_Functional_Test_7 := #_w1 AND #In_Functional_Test.Life_Trigger_PLC_Functional_Test_7;
   #Out_Functional_Test.Star_Test_PLC_Functional_Test_7 := #_w1 AND #In_Functional_Test.Star_Test_PLC_Functional_Test_7;
   #Out_Functional_Test.Button_PLC_Functional_Test_7 := #_w1 AND #In_Functional_Test.Button_PLC_Functional_Test_7;
   #Out_Functional_Test.Electrical_Current_Test_Approved_PLC_Functional_Test_7 := #_w1 AND #In_Functional_Test.Electrical_Current_Test_Approved_PLC_Functional_Test_7;
   #Out_Functional_Test.Visual_Test_Approved_PLC_Functional_Test_7 := #_w1 AND #In_Functional_Test.Visual_Test_Approved_PLC_Functional_Test_7;
   IF #_w1 THEN
       #Out_Functional_Test.Electrical_Current_Read_PLC_Functional_Test_7 := #In_Functional_Test.Electrical_Current_Read_PLC_Functional_Test_7;
   END_IF;
   #Out_Functional_Test.Life_Trigger_PLC_Functional_Test_9 := #_w1 AND #In_Functional_Test.Life_Trigger_PLC_Functional_Test_9;
   #Out_Functional_Test.Star_Test_PLC_Functional_Test_9 := #_w1 AND #In_Functional_Test.Star_Test_PLC_Functional_Test_9;
   #Out_Functional_Test.Button_PLC_Functional_Test_9 := #_w1 AND #In_Functional_Test.Button_PLC_Functional_Test_9;
   #Out_Functional_Test.Electrical_Current_Test_Approved_PLC_Functional_Test_9 := #_w1 AND #In_Functional_Test.Electrical_Current_Test_Approved_PLC_Functional_Test_9;
   #Out_Functional_Test.Visual_Test_Approved_PLC_Functional_Test_9 := #_w1 AND #In_Functional_Test.Visual_Test_Approved_PLC_Functional_Test_9;
   IF #_w1 THEN
       #Out_Functional_Test.Electrical_Current_Read_PLC_Functional_Test_9 := #In_Functional_Test.Electrical_Current_Read_PLC_Functional_Test_9;
   END_IF;
   #Out_Functional_Test.Life_Trigger_PLC_Functional_Test_11 := #_w1 AND #In_Functional_Test.Life_Trigger_PLC_Functional_Test_11;
   #Out_Functional_Test.Star_Test_PLC_Functional_Test_11 := #_w1 AND #In_Functional_Test.Star_Test_PLC_Functional_Test_11;
   #Out_Functional_Test.Button_PLC_Functional_Test_11 := #_w1 AND #In_Functional_Test.Button_PLC_Functional_Test_11;
   #Out_Functional_Test.Electrical_Current_Test_Approved_PLC_Functional_Test_11 := #_w1 AND #In_Functional_Test.Electrical_Current_Test_Approved_PLC_Functional_Test_11;
   #Out_Functional_Test.Visual_Test_Approved_PLC_Functional_Test_11 := #_w1 AND #In_Functional_Test.Visual_Test_Approved_PLC_Functional_Test_11;
   IF #_w1 THEN
       #Out_Functional_Test.Electrical_Current_Read_PLC_Functional_Test_11 := #In_Functional_Test.Electrical_Current_Read_PLC_Functional_Test_11;
   END_IF;
   #Out_Functional_Test.Life_Trigger_PLC_Functional_Test_13 := #_w1 AND #In_Functional_Test.Life_Trigger_PLC_Functional_Test_13;
   #Out_Functional_Test.Star_Test_PLC_Functional_Test_13 := #_w1 AND #In_Functional_Test.Star_Test_PLC_Functional_Test_13;
   #Out_Functional_Test.Button_PLC_Functional_Test_13 := #_w1 AND #In_Functional_Test.Button_PLC_Functional_Test_13;
   #Out_Functional_Test.Electrical_Current_Test_Approved_PLC_Functional_Test_13 := #_w1 AND #In_Functional_Test.Electrical_Current_Test_Approved_PLC_Functional_Test_13;
   #Out_Functional_Test.Visual_Test_Approved_PLC_Functional_Test_13 := #_w1 AND #In_Functional_Test.Visual_Test_Approved_PLC_Functional_Test_13;
   IF #_w1 THEN
       #Out_Functional_Test.Electrical_Current_Read_PLC_Functional_Test_13 := #In_Functional_Test.Electrical_Current_Read_PLC_Functional_Test_13;
   END_IF;
   #Out_Functional_Test.Life_Trigger_PLC_Functional_Test_15 := #_w1 AND #In_Functional_Test.Life_Trigger_PLC_Functional_Test_15;
   #Out_Functional_Test.Star_Test_PLC_Functional_Test_15 := #_w1 AND #In_Functional_Test.Star_Test_PLC_Functional_Test_15;
   #Out_Functional_Test.Button_PLC_Functional_Test_15 := #_w1 AND #In_Functional_Test.Button_PLC_Functional_Test_15;
   #Out_Functional_Test.Electrical_Current_Test_Approved_PLC_Functional_Test_15 := #_w1 AND #In_Functional_Test.Electrical_Current_Test_Approved_PLC_Functional_Test_15;
   #Out_Functional_Test.Visual_Test_Approved_PLC_Functional_Test_15 := #_w1 AND #In_Functional_Test.Visual_Test_Approved_PLC_Functional_Test_15;
   IF #_w1 THEN
       #Out_Functional_Test.Electrical_Current_Read_PLC_Functional_Test_15 := #In_Functional_Test.Electrical_Current_Read_PLC_Functional_Test_15;
   END_IF;
   #Out_Functional_Test.Life_Trigger_PLC_Functional_Test_17 := #_w1 AND #In_Functional_Test.Life_Trigger_PLC_Functional_Test_17;
   #Out_Functional_Test.Star_Test_PLC_Functional_Test_17 := #_w1 AND #In_Functional_Test.Star_Test_PLC_Functional_Test_17;
   #Out_Functional_Test.Button_PLC_Functional_Test_17 := #_w1 AND #In_Functional_Test.Button_PLC_Functional_Test_17;
   #Out_Functional_Test.Electrical_Current_Test_Approved_PLC_Functional_Test_17 := #_w1 AND #In_Functional_Test.Electrical_Current_Test_Approved_PLC_Functional_Test_17;
   #Out_Functional_Test.Visual_Test_Approved_PLC_Functional_Test_17 := #_w1 AND #In_Functional_Test.Visual_Test_Approved_PLC_Functional_Test_17;
   IF #_w1 THEN
       #Out_Functional_Test.Electrical_Current_Read_PLC_Functional_Test_17 := #In_Functional_Test.Electrical_Current_Read_PLC_Functional_Test_17;
   END_IF;
   #Out_Functional_Test.Life_Trigger_PLC_Functional_Test_19 := #_w1 AND #In_Functional_Test.Life_Trigger_PLC_Functional_Test_19;
   #Out_Functional_Test.Star_Test_PLC_Functional_Test_19 := #_w1 AND #In_Functional_Test.Star_Test_PLC_Functional_Test_19;
   #Out_Functional_Test.Button_PLC_Functional_Test_19 := #_w1 AND #In_Functional_Test.Button_PLC_Functional_Test_19;
   #Out_Functional_Test.Electrical_Current_Test_Approved_PLC_Functional_Test_19 := #_w1 AND #In_Functional_Test.Electrical_Current_Test_Approved_PLC_Functional_Test_19;
   #Out_Functional_Test.Visual_Test_Approved_PLC_Functional_Test_19 := #_w1 AND #In_Functional_Test.Visual_Test_Approved_PLC_Functional_Test_19;
   IF #_w1 THEN
       #Out_Functional_Test.Electrical_Current_Read_PLC_Functional_Test_19 := #In_Functional_Test.Electrical_Current_Read_PLC_Functional_Test_19;
   END_IF;
   #Out_Functional_Test.Life_Trigger_PLC_Functional_Test_21 := #_w1 AND #In_Functional_Test.Life_Trigger_PLC_Functional_Test_21;
   #Out_Functional_Test.Star_Test_PLC_Functional_Test_21 := #_w1 AND #In_Functional_Test.Star_Test_PLC_Functional_Test_21;
   #Out_Functional_Test.Button_PLC_Functional_Test_21 := #_w1 AND #In_Functional_Test.Button_PLC_Functional_Test_21;
   #Out_Functional_Test.Electrical_Current_Test_Approved_PLC_Functional_Test_21 := #_w1 AND #In_Functional_Test.Electrical_Current_Test_Approved_PLC_Functional_Test_21;
   #Out_Functional_Test.Visual_Test_Approved_PLC_Functional_Test_21 := #_w1 AND #In_Functional_Test.Visual_Test_Approved_PLC_Functional_Test_21;
   IF #_w1 THEN
       #Out_Functional_Test.Electrical_Current_Read_PLC_Functional_Test_21 := #In_Functional_Test.Electrical_Current_Read_PLC_Functional_Test_21;
   END_IF;
   #Out_Functional_Test.Life_Trigger_PLC_Functional_Test_23 := #_w1 AND #In_Functional_Test.Life_Trigger_PLC_Functional_Test_23;
   #Out_Functional_Test.Star_Test_PLC_Functional_Test_23 := #_w1 AND #In_Functional_Test.Star_Test_PLC_Functional_Test_23;
   #Out_Functional_Test.Button_PLC_Functional_Test_23 := #_w1 AND #In_Functional_Test.Button_PLC_Functional_Test_23;
   #Out_Functional_Test.Electrical_Current_Test_Approved_PLC_Functional_Test_23 := #_w1 AND #In_Functional_Test.Electrical_Current_Test_Approved_PLC_Functional_Test_23;
   #Out_Functional_Test.Visual_Test_Approved_PLC_Functional_Test_23 := #_w1 AND #In_Functional_Test.Visual_Test_Approved_PLC_Functional_Test_23;
   IF #_w1 THEN
       #Out_Functional_Test.Electrical_Current_Read_PLC_Functional_Test_23 := #In_Functional_Test.Electrical_Current_Read_PLC_Functional_Test_23;
   END_IF;
   #Out_Functional_Test.Life_Trigger_PLC_Functional_Test_25 := #_w1 AND #In_Functional_Test.Life_Trigger_PLC_Functional_Test_25;
   #Out_Functional_Test.Star_Test_PLC_Functional_Test_25 := #_w1 AND #In_Functional_Test.Star_Test_PLC_Functional_Test_25;
   #Out_Functional_Test.Button_PLC_Functional_Test_25 := #_w1 AND #In_Functional_Test.Button_PLC_Functional_Test_25;
   #Out_Functional_Test.Electrical_Current_Test_Approved_PLC_Functional_Test_25 := #_w1 AND #In_Functional_Test.Electrical_Current_Test_Approved_PLC_Functional_Test_25;
   #Out_Functional_Test.Visual_Test_Approved_PLC_Functional_Test_25 := #_w1 AND #In_Functional_Test.Visual_Test_Approved_PLC_Functional_Test_25;
   IF #_w1 THEN
       #Out_Functional_Test.Electrical_Current_Read_PLC_Functional_Test_25 := #In_Functional_Test.Electrical_Current_Read_PLC_Functional_Test_25;
   END_IF;
   #Out_Functional_Test.Life_Trigger_PLC_Functional_Test_27 := #_w1 AND #In_Functional_Test.Life_Trigger_PLC_Functional_Test_27;
   #Out_Functional_Test.Star_Test_PLC_Functional_Test_27 := #_w1 AND #In_Functional_Test.Star_Test_PLC_Functional_Test_27;
   #Out_Functional_Test.Button_PLC_Functional_Test_27 := #_w1 AND #In_Functional_Test.Button_PLC_Functional_Test_27;
   #Out_Functional_Test.Electrical_Current_Test_Approved_PLC_Functional_Test_27 := #_w1 AND #In_Functional_Test.Electrical_Current_Test_Approved_PLC_Functional_Test_27;
   #Out_Functional_Test.Visual_Test_Approved_PLC_Functional_Test_27 := #_w1 AND #In_Functional_Test.Visual_Test_Approved_PLC_Functional_Test_27;
   IF #_w1 THEN
       #Out_Functional_Test.Electrical_Current_Read_PLC_Functional_Test_27 := #In_Functional_Test.Electrical_Current_Read_PLC_Functional_Test_27;
   END_IF;
   #Out_Functional_Test.Life_Trigger_PLC_Functional_Test_29 := #_w1 AND #In_Functional_Test.Life_Trigger_PLC_Functional_Test_29;
   #Out_Functional_Test.Star_Test_PLC_Functional_Test_29 := #_w1 AND #In_Functional_Test.Star_Test_PLC_Functional_Test_29;
   #Out_Functional_Test.Button_PLC_Functional_Test_29 := #_w1 AND #In_Functional_Test.Button_PLC_Functional_Test_29;
   #Out_Functional_Test.Electrical_Current_Test_Approved_PLC_Functional_Test_29 := #_w1 AND #In_Functional_Test.Electrical_Current_Test_Approved_PLC_Functional_Test_29;
   #Out_Functional_Test.Visual_Test_Approved_PLC_Functional_Test_29 := #_w1 AND #In_Functional_Test.Visual_Test_Approved_PLC_Functional_Test_29;
   IF #_w1 THEN
       #Out_Functional_Test.Electrical_Current_Read_PLC_Functional_Test_29 := #In_Functional_Test.Electrical_Current_Read_PLC_Functional_Test_29;
   END_IF;
END_REGION

REGION Network 5: Functional Test Station 7
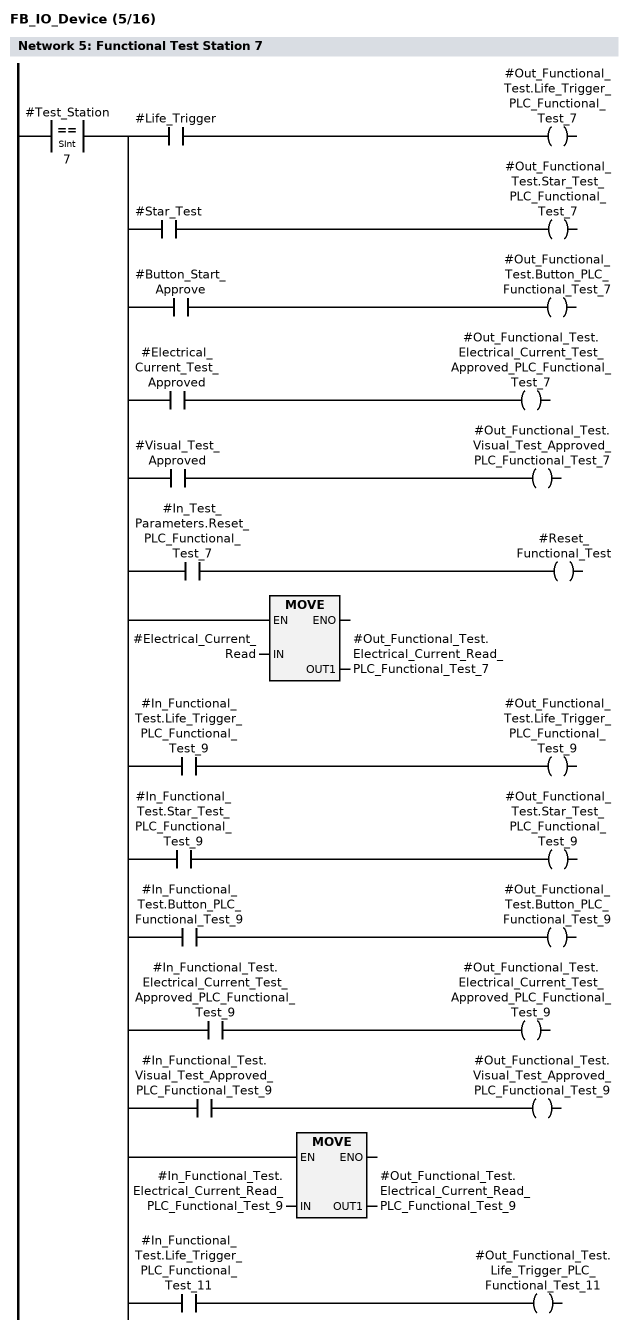
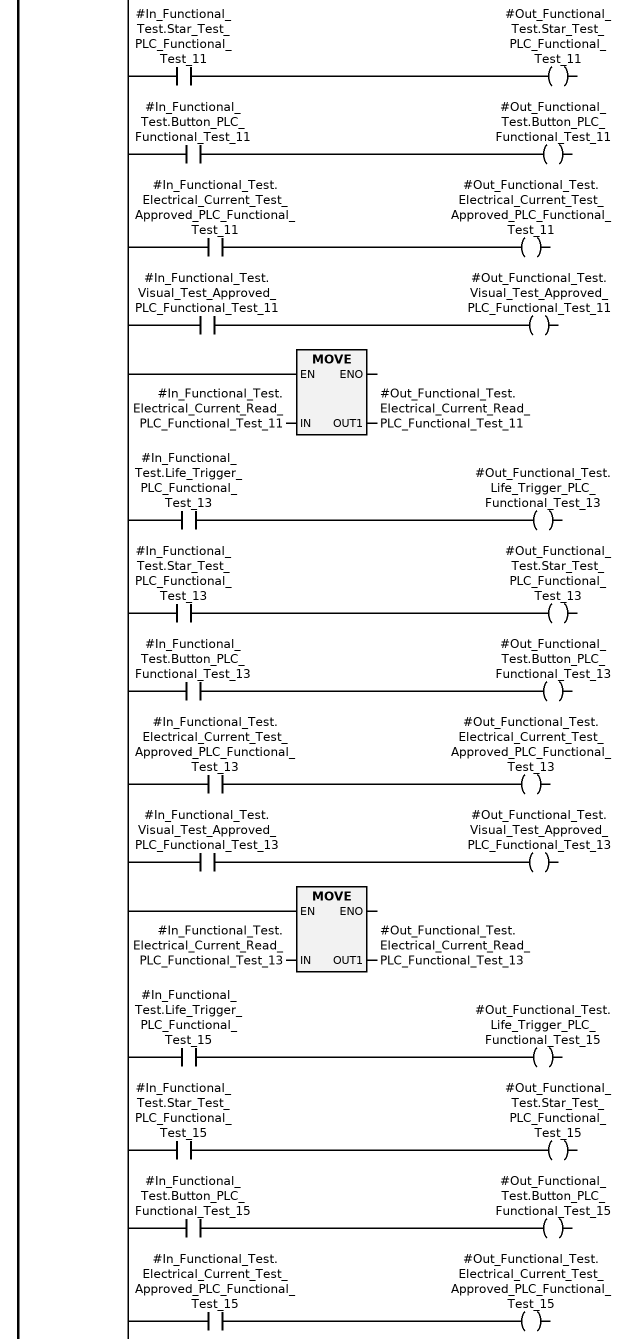
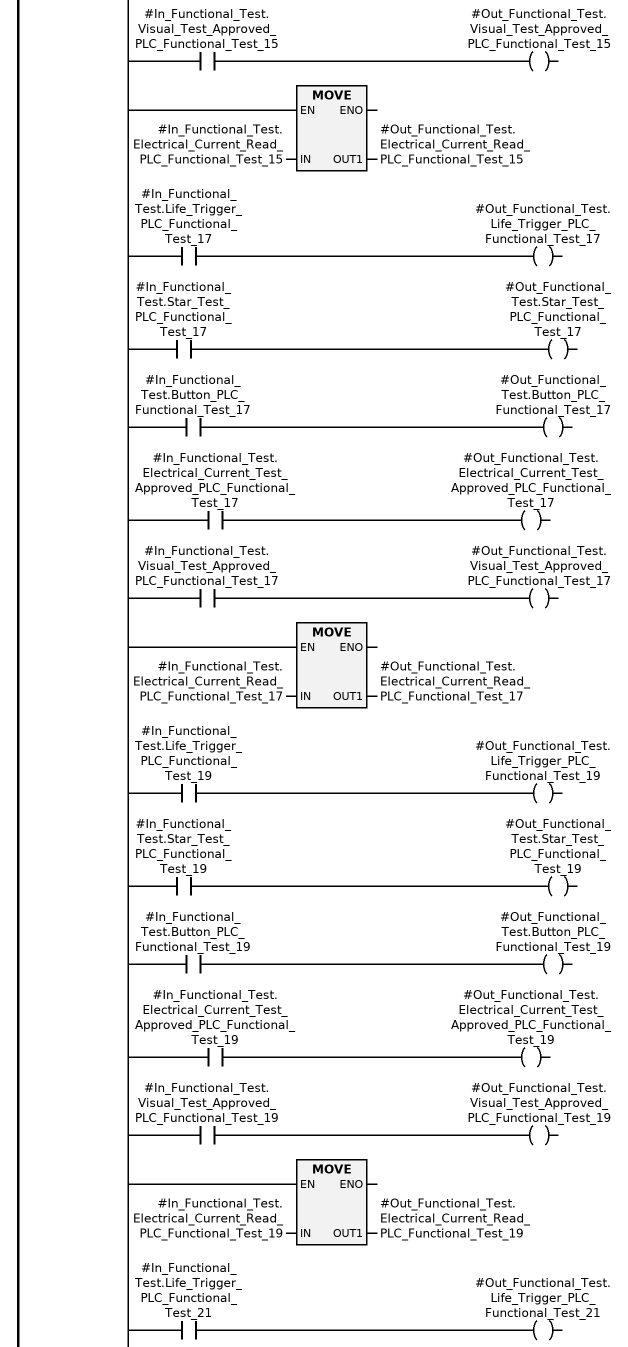
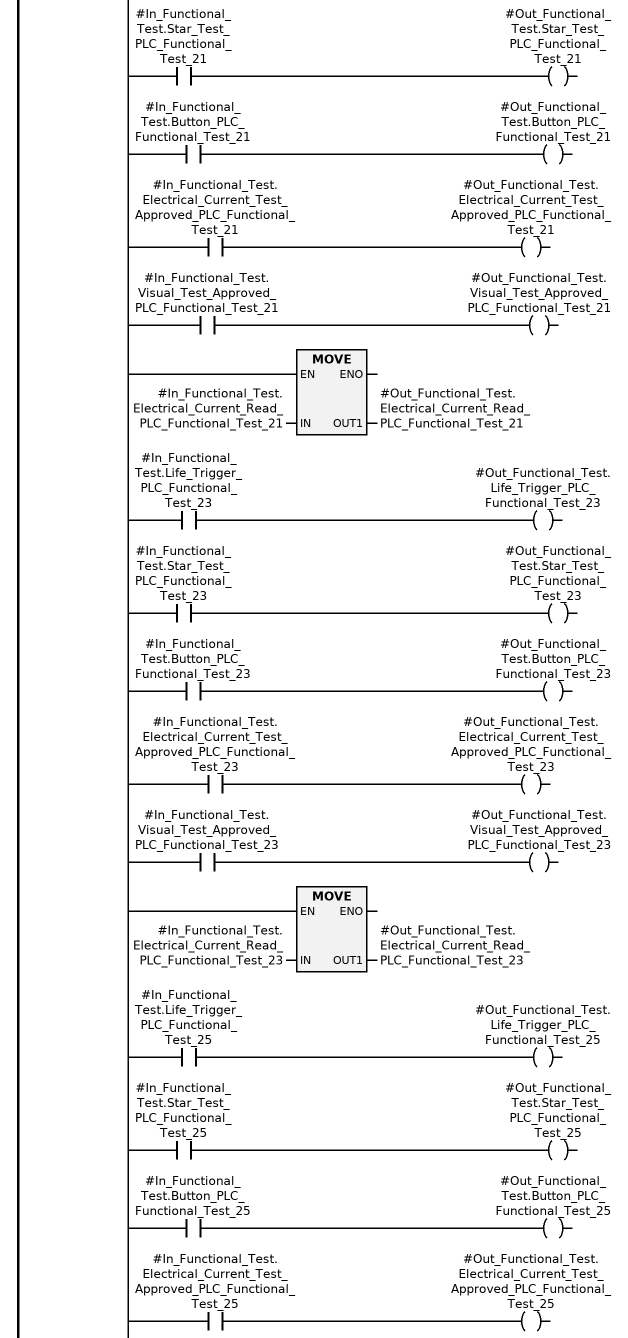
